//     Drive/Outputs/Out/nCtrl1 @bit 2 <-> STM Control/Control/Reduce torque
//     Drive/Outputs/Out/nCtrl1 @bit 1 <-> STM Control/Control/Reset
//     Drive/Outputs/Out/nDataOut2[0] <-> STM Velocity/Velocity
//   (this object) <-> Device 1 (EtherCAT)/Power (EK1200)/PLC Junction 2 (EK1122)/PLC Coupler 2 (EK1100)/PLC Junction 10 (EK1122)/Granite3 (EK1100)/PLC Junction 12  (EK1122)/TM2K4 (EK1100)/TM2K4-EL5042-E3
//     Enc/Inputs/In/nComState @bit 1 <-> WcState/InputToggle
//     Enc/Inputs/In/nComState <-> WcState/WcState
//     Enc/Inputs/In/nDataIn1 <-> FB Inputs Channel 1/Position
//     Enc/Inputs/In/nDataIn1 <-> FB Inputs Channel 2/Position
//     Enc/Inputs/In/nState1 @bit 12 <-> FB Inputs Channel 1/Status/Diag
//     Enc/Inputs/In/nState1 @bit 12 <-> FB Inputs Channel 2/Status/Diag
//     Enc/Inputs/In/nState1 @bit 1 <-> FB Inputs Channel 1/Status/Error
//     Enc/Inputs/In/nState1 @bit 1 <-> FB Inputs Channel 2/Status/Error
//     Enc/Inputs/In/nState1 @bit 14 <-> FB Inputs Channel 1/Status/Input cycle counter
//     Enc/Inputs/In/nState1 @bit 14 <-> FB Inputs Channel 2/Status/Input cycle counter
//     Enc/Inputs/In/nState1 @bit 2 <-> FB Inputs Channel 1/Status/Ready
//     Enc/Inputs/In/nState1 @bit 2 <-> FB Inputs Channel 2/Status/Ready
//     Enc/Inputs/In/nState1 @bit 13 <-> FB Inputs Channel 1/Status/TxPDO State
//     Enc/Inputs/In/nState1 @bit 13 <-> FB Inputs Channel 2/Status/TxPDO State
//     Enc/Inputs/In/nState1 <-> FB Inputs Channel 1/Status/Warning
//     Enc/Inputs/In/nState1 <-> FB Inputs Channel 2/Status/Warning
//   (this object) <-> Device 1 (EtherCAT)/Power (EK1200)/PLC Junction 2 (EK1122)/PLC Coupler 2 (EK1100)/PLC Junction 10 (EK1122)/Granite3 (EK1100)/PLC Junction 12  (EK1122)/TM2K4 (EK1100)/TM2K4-EL7041-E1
//     Drive/Inputs/In/nState1 @bit 3 <-> STM Status/Status/Error
//     Drive/Inputs/In/nState1 @bit 5 <-> STM Status/Status/Moving negative
//     Drive/Inputs/In/nState1 @bit 4 <-> STM Status/Status/Moving positive
//     Drive/Inputs/In/nState1 @bit 1 <-> STM Status/Status/Ready
//     Drive/Inputs/In/nState1 <-> STM Status/Status/Ready to enable
//     Drive/Inputs/In/nState1 @bit 6 <-> STM Status/Status/Torque reduced
//     Drive/Inputs/In/nState1 @bit 2 <-> STM Status/Status/Warning
//     Drive/Inputs/In/nState2 @bit 3 <-> STM Status/Status/Digital input 1
//     Drive/Inputs/In/nState2 @bit 4 <-> STM Status/Status/Digital input 2
//     Drive/Inputs/In/nState2 @bit 5 <-> STM Status/Status/Sync error
//     Drive/Inputs/In/nState2 @bit 7 <-> STM Status/Status/TxPDO Toggle
//     Drive/Inputs/In/nState4 @bit 1 <-> WcState/InputToggle
//     Drive/Inputs/In/nState4 <-> WcState/WcState
//     Drive/Outputs/Out/nCtrl1 <-> STM Control/Control/Enable
//     Drive/Outputs/Out/nCtrl1 @bit 2 <-> STM Control/Control/Reduce torque
//     Drive/Outputs/Out/nCtrl1 @bit 1 <-> STM Control/Control/Reset
//     Drive/Outputs/Out/nDataOut2[0] <-> STM Velocity/Velocity
//   (this object) <-> Device 1 (EtherCAT)/Power (EK1200)/PLC Junction 2 (EK1122)/PLC Coupler 2 (EK1100)/PLC Junction 10 (EK1122)/Granite3 (EK1100)/PLC Junction 12  (EK1122)/TM2K4 (EK1100)/TM2K4-EL7041-E2
//     Drive/Inputs/In/nState1 @bit 3 <-> STM Status/Status/Error
//     Drive/Inputs/In/nState1 @bit 5 <-> STM Status/Status/Moving negative
//     Drive/Inputs/In/nState1 @bit 4 <-> STM Status/Status/Moving positive
//     Drive/Inputs/In/nState1 @bit 1 <-> STM Status/Status/Ready
//     Drive/Inputs/In/nState1 <-> STM Status/Status/Ready to enable
//     Drive/Inputs/In/nState1 @bit 6 <-> STM Status/Status/Torque reduced
//     Drive/Inputs/In/nState1 @bit 2 <-> STM Status/Status/Warning
//     Drive/Inputs/In/nState2 @bit 3 <-> STM Status/Status/Digital input 1
//     Drive/Inputs/In/nState2 @bit 4 <-> STM Status/Status/Digital input 2
//     Drive/Inputs/In/nState2 @bit 5 <-> STM Status/Status/Sync error
//     Drive/Inputs/In/nState2 @bit 7 <-> STM Status/Status/TxPDO Toggle
//     Drive/Inputs/In/nState4 @bit 1 <-> WcState/InputToggle
//     Drive/Inputs/In/nState4 <-> WcState/WcState
//     Drive/Outputs/Out/nCtrl1 <-> STM Control/Control/Enable
//     Drive/Outputs/Out/nCtrl1 @bit 2 <-> STM Control/Control/Reduce torque
//     Drive/Outputs/Out/nCtrl1 @bit 1 <-> STM Control/Control/Reset
//     Drive/Outputs/Out/nDataOut2[0] <-> STM Velocity/Velocity
//   (this object) <-> Device 1 (EtherCAT)/Power (EK1200)/PLC Junction 2 (EK1122)/PLC Coupler 2 (EK1100)/PLC Junction 10 (EK1122)/Granite3 (EK1100)/PLC Junction 12  (EK1122)/IM6K4 (EK1100)/IM6K4-EL5042-E2
//     Enc/Inputs/In/nComState @bit 1 <-> WcState/InputToggle
//     Enc/Inputs/In/nComState <-> WcState/WcState
//     Enc/Inputs/In/nDataIn1 <-> FB Inputs Channel 1/Position
//     Enc/Inputs/In/nState1 @bit 12 <-> FB Inputs Channel 1/Status/Diag
//     Enc/Inputs/In/nState1 @bit 1 <-> FB Inputs Channel 1/Status/Error
//     Enc/Inputs/In/nState1 @bit 14 <-> FB Inputs Channel 1/Status/Input cycle counter
//     Enc/Inputs/In/nState1 @bit 2 <-> FB Inputs Channel 1/Status/Ready
//     Enc/Inputs/In/nState1 @bit 13 <-> FB Inputs Channel 1/Status/TxPDO State
//     Enc/Inputs/In/nState1 <-> FB Inputs Channel 1/Status/Warning
//   (this object) <-> Device 1 (EtherCAT)/Power (EK1200)/PLC Junction 2 (EK1122)/PLC Coupler 2 (EK1100)/PLC Junction 10 (EK1122)/Granite3 (EK1100)/PLC Junction 12  (EK1122)/IM6K4 (EK1100)/IM6K4-EL7041-E1
//     Drive/Inputs/In/nState1 @bit 3 <-> STM Status/Status/Error
//     Drive/Inputs/In/nState1 @bit 5 <-> STM Status/Status/Moving negative
//     Drive/Inputs/In/nState1 @bit 4 <-> STM Status/Status/Moving positive
//     Drive/Inputs/In/nState1 @bit 1 <-> STM Status/Status/Ready
//     Drive/Inputs/In/nState1 <-> STM Status/Status/Ready to enable
//     Drive/Inputs/In/nState1 @bit 6 <-> STM Status/Status/Torque reduced
//     Drive/Inputs/In/nState1 @bit 2 <-> STM Status/Status/Warning
//     Drive/Inputs/In/nState2 @bit 3 <-> STM Status/Status/Digital input 1
//     Drive/Inputs/In/nState2 @bit 4 <-> STM Status/Status/Digital input 2
//     Drive/Inputs/In/nState2 @bit 5 <-> STM Status/Status/Sync error
//     Drive/Inputs/In/nState2 @bit 7 <-> STM Status/Status/TxPDO Toggle
//     Drive/Inputs/In/nState4 @bit 1 <-> WcState/InputToggle
//     Drive/Inputs/In/nState4 <-> WcState/WcState
//     Drive/Outputs/Out/nCtrl1 <-> STM Control/Control/Enable
//     Drive/Outputs/Out/nCtrl1 @bit 2 <-> STM Control/Control/Reduce torque
//     Drive/Outputs/Out/nCtrl1 @bit 1 <-> STM Control/Control/Reset
//     Drive/Outputs/Out/nDataOut2[0] <-> STM Velocity/Velocity
//   (this object) <-> Device 1 (EtherCAT)/Power (EK1200)/PLC Junction 2 (EK1122)/PLC Coupler 2 (EK1100)/PLC Junction 10 (EK1122)/Granite3 (EK1100)/PLC Junction 11 (EK1122)/PF2K4-WFS (EK1100)/PF2K4-EL5042-E3
//     Enc/Inputs/In/nComState @bit 1 <-> WcState/InputToggle
//     Enc/Inputs/In/nComState <-> WcState/WcState
//     Enc/Inputs/In/nDataIn1 <-> FB Inputs Channel 2/Position
//     Enc/Inputs/In/nDataIn1 <-> FB Inputs Channel 1/Position
//     Enc/Inputs/In/nState1 @bit 12 <-> FB Inputs Channel 2/Status/Diag
//     Enc/Inputs/In/nState1 @bit 12 <-> FB Inputs Channel 1/Status/Diag
//     Enc/Inputs/In/nState1 @bit 1 <-> FB Inputs Channel 2/Status/Error
//     Enc/Inputs/In/nState1 @bit 1 <-> FB Inputs Channel 1/Status/Error
//     Enc/Inputs/In/nState1 @bit 14 <-> FB Inputs Channel 2/Status/Input cycle counter
//     Enc/Inputs/In/nState1 @bit 14 <-> FB Inputs Channel 1/Status/Input cycle counter
//     Enc/Inputs/In/nState1 @bit 2 <-> FB Inputs Channel 2/Status/Ready
//     Enc/Inputs/In/nState1 @bit 2 <-> FB Inputs Channel 1/Status/Ready
//     Enc/Inputs/In/nState1 @bit 13 <-> FB Inputs Channel 2/Status/TxPDO State
//     Enc/Inputs/In/nState1 @bit 13 <-> FB Inputs Channel 1/Status/TxPDO State
//     Enc/Inputs/In/nState1 <-> FB Inputs Channel 2/Status/Warning
//     Enc/Inputs/In/nState1 <-> FB Inputs Channel 1/Status/Warning
//   (this object) <-> Device 1 (EtherCAT)/Power (EK1200)/PLC Junction 2 (EK1122)/PLC Coupler 2 (EK1100)/PLC Junction 10 (EK1122)/Granite3 (EK1100)/PLC Junction 11 (EK1122)/PF2K4-WFS (EK1100)/PF2K4-EL7041-E1
//     Drive/Inputs/In/nState1 @bit 3 <-> STM Status/Status/Error
//     Drive/Inputs/In/nState1 @bit 5 <-> STM Status/Status/Moving negative
//     Drive/Inputs/In/nState1 @bit 4 <-> STM Status/Status/Moving positive
//     Drive/Inputs/In/nState1 @bit 1 <-> STM Status/Status/Ready
//     Drive/Inputs/In/nState1 <-> STM Status/Status/Ready to enable
//     Drive/Inputs/In/nState1 @bit 6 <-> STM Status/Status/Torque reduced
//     Drive/Inputs/In/nState1 @bit 2 <-> STM Status/Status/Warning
//     Drive/Inputs/In/nState2 @bit 3 <-> STM Status/Status/Digital input 1
//     Drive/Inputs/In/nState2 @bit 4 <-> STM Status/Status/Digital input 2
//     Drive/Inputs/In/nState2 @bit 5 <-> STM Status/Status/Sync error
//     Drive/Inputs/In/nState2 @bit 7 <-> STM Status/Status/TxPDO Toggle
//     Drive/Inputs/In/nState4 @bit 1 <-> WcState/InputToggle
//     Drive/Inputs/In/nState4 <-> WcState/WcState
//     Drive/Outputs/Out/nCtrl1 <-> STM Control/Control/Enable
//     Drive/Outputs/Out/nCtrl1 @bit 2 <-> STM Control/Control/Reduce torque
//     Drive/Outputs/Out/nCtrl1 @bit 1 <-> STM Control/Control/Reset
//     Drive/Outputs/Out/nDataOut2[0] <-> STM Velocity/Velocity
//   (this object) <-> Device 1 (EtherCAT)/Power (EK1200)/PLC Junction 2 (EK1122)/PLC Coupler 2 (EK1100)/PLC Junction 10 (EK1122)/Granite3 (EK1100)/PLC Junction 11 (EK1122)/PF2K4-WFS (EK1100)/PF2K4-EL7041-E2
//     Drive/Inputs/In/nState1 @bit 3 <-> STM Status/Status/Error
//     Drive/Inputs/In/nState1 @bit 5 <-> STM Status/Status/Moving negative
//     Drive/Inputs/In/nState1 @bit 4 <-> STM Status/Status/Moving positive
//     Drive/Inputs/In/nState1 @bit 1 <-> STM Status/Status/Ready
//     Drive/Inputs/In/nState1 <-> STM Status/Status/Ready to enable
//     Drive/Inputs/In/nState1 @bit 6 <-> STM Status/Status/Torque reduced
//     Drive/Inputs/In/nState1 @bit 2 <-> STM Status/Status/Warning
//     Drive/Inputs/In/nState2 @bit 3 <-> STM Status/Status/Digital input 1
//     Drive/Inputs/In/nState2 @bit 4 <-> STM Status/Status/Digital input 2
//     Drive/Inputs/In/nState2 @bit 5 <-> STM Status/Status/Sync error
//     Drive/Inputs/In/nState2 @bit 7 <-> STM Status/Status/TxPDO Toggle
//     Drive/Inputs/In/nState4 @bit 1 <-> WcState/InputToggle
//     Drive/Inputs/In/nState4 <-> WcState/WcState
//     Drive/Outputs/Out/nCtrl1 <-> STM Control/Control/Enable
//     Drive/Outputs/Out/nCtrl1 @bit 2 <-> STM Control/Control/Reduce torque
//     Drive/Outputs/Out/nCtrl1 @bit 1 <-> STM Control/Control/Reset
//     Drive/Outputs/Out/nDataOut2[0] <-> STM Velocity/Velocity
//   (this object) <-> Device 1 (EtherCAT)/Power (EK1200)/PLC Junction 2 (EK1122)/PLC Coupler 2 (EK1100)/PLC Junction 9 (EK1122)/SP1K4 Bottom Rail (EK1100)/EL7031-LensX
//     Drive/Inputs/In/nState1 @bit 3 <-> STM Status/Status/Error
//     Drive/Inputs/In/nState1 @bit 5 <-> STM Status/Status/Moving negative
//     Drive/Inputs/In/nState1 @bit 4 <-> STM Status/Status/Moving positive
//     Drive/Inputs/In/nState1 @bit 1 <-> STM Status/Status/Ready
//     Drive/Inputs/In/nState1 <-> STM Status/Status/Ready to enable
//     Drive/Inputs/In/nState1 @bit 6 <-> STM Status/Status/Torque reduced
//     Drive/Inputs/In/nState1 @bit 2 <-> STM Status/Status/Warning
//     Drive/Inputs/In/nState2 @bit 3 <-> STM Status/Status/Digital input 1
//     Drive/Inputs/In/nState2 @bit 4 <-> STM Status/Status/Digital input 2
//     Drive/Inputs/In/nState2 @bit 5 <-> STM Status/Status/Sync error
//     Drive/Inputs/In/nState2 @bit 7 <-> STM Status/Status/TxPDO Toggle
//     Drive/Inputs/In/nState4 @bit 1 <-> WcState/InputToggle
//     Drive/Inputs/In/nState4 <-> WcState/WcState
//     Drive/Outputs/Out/nCtrl1 <-> STM Control/Control/Enable
//     Drive/Outputs/Out/nCtrl1 @bit 2 <-> STM Control/Control/Reduce torque
//     Drive/Outputs/Out/nCtrl1 @bit 1 <-> STM Control/Control/Reset
//     Drive/Outputs/Out/nDataOut2[0] <-> STM Velocity/Velocity
//     Enc/Inputs/In/nDataIn1[0] <-> ENC Status compact/Counter value
//     Enc/Inputs/In/nDataIn2[0] <-> ENC Status compact/Latch value
//     Enc/Inputs/In/nState1 @bit 4 <-> ENC Status compact/Status/Counter overflow
//     Enc/Inputs/In/nState1 @bit 3 <-> ENC Status compact/Status/Counter underflow
//     Enc/Inputs/In/nState1 @bit 1 <-> ENC Status compact/Status/Latch extern valid
//     Enc/Inputs/In/nState1 @bit 2 <-> ENC Status compact/Status/Set counter done
//     Enc/Inputs/In/nState2 @bit 4 <-> ENC Status compact/Status/Status of extern latch
//     Enc/Inputs/In/nState2 @bit 5 <-> ENC Status compact/Status/Sync error
//     Enc/Inputs/In/nState2 @bit 7 <-> ENC Status compact/Status/TxPDO Toggle
//     Enc/Inputs/In/nState4 @bit 1 <-> WcState/InputToggle
//     Enc/Inputs/In/nState4 <-> WcState/WcState
//     Enc/Outputs/Out/nCtrl1 @bit 3 <-> ENC Control compact/Control/Enable latch extern on negative edge
//     Enc/Outputs/Out/nCtrl1 @bit 1 <-> ENC Control compact/Control/Enable latch extern on positive edge
//     Enc/Outputs/Out/nCtrl1 @bit 2 <-> ENC Control compact/Control/Set counter
//     Enc/Outputs/Out/nDataOut1[0] <-> ENC Control compact/Set counter value
//   (this object) <-> Device 1 (EtherCAT)/Power (EK1200)/PLC Junction 2 (EK1122)/PLC Coupler 2 (EK1100)/PLC Junction 9 (EK1122)/SP1K4 Bottom Rail (EK1100)/FoilX-EL7041
//     Drive/Inputs/In/nState1 @bit 3 <-> STM Status/Status/Error
//     Drive/Inputs/In/nState1 @bit 5 <-> STM Status/Status/Moving negative
//     Drive/Inputs/In/nState1 @bit 4 <-> STM Status/Status/Moving positive
//     Drive/Inputs/In/nState1 @bit 1 <-> STM Status/Status/Ready
//     Drive/Inputs/In/nState1 <-> STM Status/Status/Ready to enable
//     Drive/Inputs/In/nState1 @bit 6 <-> STM Status/Status/Torque reduced
//     Drive/Inputs/In/nState1 @bit 2 <-> STM Status/Status/Warning
//     Drive/Inputs/In/nState2 @bit 3 <-> STM Status/Status/Digital input 1
//     Drive/Inputs/In/nState2 @bit 4 <-> STM Status/Status/Digital input 2
//     Drive/Inputs/In/nState2 @bit 5 <-> STM Status/Status/Sync error
//     Drive/Inputs/In/nState2 @bit 7 <-> STM Status/Status/TxPDO Toggle
//     Drive/Inputs/In/nState4 @bit 1 <-> WcState/InputToggle
//     Drive/Inputs/In/nState4 <-> WcState/WcState
//     Drive/Outputs/Out/nCtrl1 <-> STM Control/Control/Enable
//     Drive/Outputs/Out/nCtrl1 @bit 2 <-> STM Control/Control/Reduce torque
//     Drive/Outputs/Out/nCtrl1 @bit 1 <-> STM Control/Control/Reset
//     Drive/Outputs/Out/nDataOut2[0] <-> STM Velocity/Velocity
//   (this object) <-> Device 1 (EtherCAT)/Power (EK1200)/PLC Junction 2 (EK1122)/PLC Coupler 2 (EK1100)/PLC Junction 9 (EK1122)/SP1K4 Top Rail (EK1100)/SP1K4-EL5042-E2
//     Enc/Inputs/In/nComState @bit 1 <-> WcState/InputToggle
//     Enc/Inputs/In/nComState <-> WcState/WcState
//     Enc/Inputs/In/nDataIn1 <-> FB Inputs Channel 2/Position
//     Enc/Inputs/In/nDataIn1 <-> FB Inputs Channel 1/Position
//     Enc/Inputs/In/nState1 @bit 12 <-> FB Inputs Channel 2/Status/Diag
//     Enc/Inputs/In/nState1 @bit 12 <-> FB Inputs Channel 1/Status/Diag
//     Enc/Inputs/In/nState1 @bit 1 <-> FB Inputs Channel 2/Status/Error
//     Enc/Inputs/In/nState1 @bit 1 <-> FB Inputs Channel 1/Status/Error
//     Enc/Inputs/In/nState1 @bit 14 <-> FB Inputs Channel 2/Status/Input cycle counter
//     Enc/Inputs/In/nState1 @bit 14 <-> FB Inputs Channel 1/Status/Input cycle counter
//     Enc/Inputs/In/nState1 @bit 2 <-> FB Inputs Channel 2/Status/Ready
//     Enc/Inputs/In/nState1 @bit 2 <-> FB Inputs Channel 1/Status/Ready
//     Enc/Inputs/In/nState1 @bit 13 <-> FB Inputs Channel 2/Status/TxPDO State
//     Enc/Inputs/In/nState1 @bit 13 <-> FB Inputs Channel 1/Status/TxPDO State
//     Enc/Inputs/In/nState1 <-> FB Inputs Channel 2/Status/Warning
//     Enc/Inputs/In/nState1 <-> FB Inputs Channel 1/Status/Warning
//   (this object) <-> Device 1 (EtherCAT)/Power (EK1200)/PLC Junction 2 (EK1122)/PLC Coupler 2 (EK1100)/PLC Junction 9 (EK1122)/SP1K4 Bottom Rail (EK1100)/ZonePlateX-EL7041
//     Drive/Inputs/In/nState1 @bit 3 <-> STM Status/Status/Error
//     Drive/Inputs/In/nState1 @bit 5 <-> STM Status/Status/Moving negative
//     Drive/Inputs/In/nState1 @bit 4 <-> STM Status/Status/Moving positive
//     Drive/Inputs/In/nState1 @bit 1 <-> STM Status/Status/Ready
//     Drive/Inputs/In/nState1 <-> STM Status/Status/Ready to enable
//     Drive/Inputs/In/nState1 @bit 6 <-> STM Status/Status/Torque reduced
//     Drive/Inputs/In/nState1 @bit 2 <-> STM Status/Status/Warning
//     Drive/Inputs/In/nState2 @bit 3 <-> STM Status/Status/Digital input 1
//     Drive/Inputs/In/nState2 @bit 4 <-> STM Status/Status/Digital input 2
//     Drive/Inputs/In/nState2 @bit 5 <-> STM Status/Status/Sync error
//     Drive/Inputs/In/nState2 @bit 7 <-> STM Status/Status/TxPDO Toggle
//     Drive/Inputs/In/nState4 @bit 1 <-> WcState/InputToggle
//     Drive/Inputs/In/nState4 <-> WcState/WcState
//     Drive/Outputs/Out/nCtrl1 <-> STM Control/Control/Enable
//     Drive/Outputs/Out/nCtrl1 @bit 2 <-> STM Control/Control/Reduce torque
//     Drive/Outputs/Out/nCtrl1 @bit 1 <-> STM Control/Control/Reset
//     Drive/Outputs/Out/nDataOut2[0] <-> STM Velocity/Velocity
//   (this object) <-> Device 1 (EtherCAT)/Power (EK1200)/PLC Junction 2 (EK1122)/PLC Coupler 2 (EK1100)/PLC Junction 9 (EK1122)/SP1K4 Top Rail (EK1100)/SP1K4-EL5042-E1
//     Enc/Inputs/In/nComState @bit 1 <-> WcState/InputToggle
//     Enc/Inputs/In/nComState <-> WcState/WcState
//     Enc/Inputs/In/nDataIn1 <-> FB Inputs Channel 1/Position
//     Enc/Inputs/In/nDataIn1 <-> FB Inputs Channel 2/Position
//     Enc/Inputs/In/nState1 @bit 12 <-> FB Inputs Channel 1/Status/Diag
//     Enc/Inputs/In/nState1 @bit 12 <-> FB Inputs Channel 2/Status/Diag
//     Enc/Inputs/In/nState1 @bit 1 <-> FB Inputs Channel 1/Status/Error
//     Enc/Inputs/In/nState1 @bit 1 <-> FB Inputs Channel 2/Status/Error
//     Enc/Inputs/In/nState1 @bit 14 <-> FB Inputs Channel 1/Status/Input cycle counter
//     Enc/Inputs/In/nState1 @bit 14 <-> FB Inputs Channel 2/Status/Input cycle counter
//     Enc/Inputs/In/nState1 @bit 2 <-> FB Inputs Channel 1/Status/Ready
//     Enc/Inputs/In/nState1 @bit 2 <-> FB Inputs Channel 2/Status/Ready
//     Enc/Inputs/In/nState1 @bit 13 <-> FB Inputs Channel 1/Status/TxPDO State
//     Enc/Inputs/In/nState1 @bit 13 <-> FB Inputs Channel 2/Status/TxPDO State
//     Enc/Inputs/In/nState1 <-> FB Inputs Channel 1/Status/Warning
//     Enc/Inputs/In/nState1 <-> FB Inputs Channel 2/Status/Warning
//   (this object) <-> Device 1 (EtherCAT)/Power (EK1200)/PLC Junction 2 (EK1122)/PLC Coupler 2 (EK1100)/PLC Junction 9 (EK1122)/SP1K4 Bottom Rail (EK1100)/ZonePlateY-EL7041
//     Drive/Inputs/In/nState1 @bit 3 <-> STM Status/Status/Error
//     Drive/Inputs/In/nState1 @bit 5 <-> STM Status/Status/Moving negative
//     Drive/Inputs/In/nState1 @bit 4 <-> STM Status/Status/Moving positive
//     Drive/Inputs/In/nState1 @bit 1 <-> STM Status/Status/Ready
//     Drive/Inputs/In/nState1 <-> STM Status/Status/Ready to enable
//     Drive/Inputs/In/nState1 @bit 6 <-> STM Status/Status/Torque reduced
//     Drive/Inputs/In/nState1 @bit 2 <-> STM Status/Status/Warning
//     Drive/Inputs/In/nState2 @bit 3 <-> STM Status/Status/Digital input 1
//     Drive/Inputs/In/nState2 @bit 4 <-> STM Status/Status/Digital input 2
//     Drive/Inputs/In/nState2 @bit 5 <-> STM Status/Status/Sync error
//     Drive/Inputs/In/nState2 @bit 7 <-> STM Status/Status/TxPDO Toggle
//     Drive/Inputs/In/nState4 @bit 1 <-> WcState/InputToggle
//     Drive/Inputs/In/nState4 <-> WcState/WcState
//     Drive/Outputs/Out/nCtrl1 <-> STM Control/Control/Enable
//     Drive/Outputs/Out/nCtrl1 @bit 2 <-> STM Control/Control/Reduce torque
//     Drive/Outputs/Out/nCtrl1 @bit 1 <-> STM Control/Control/Reset
//     Drive/Outputs/Out/nDataOut2[0] <-> STM Velocity/Velocity
//   (this object) <-> Device 1 (EtherCAT)/Power (EK1200)/PLC Junction 2 (EK1122)/PLC Coupler 2 (EK1100)/PLC Junction 9 (EK1122)/SP1K4 Bottom Rail (EK1100)/ZonePlateZ-EL7041
//     Drive/Inputs/In/nState1 @bit 3 <-> STM Status/Status/Error
//     Drive/Inputs/In/nState1 @bit 5 <-> STM Status/Status/Moving negative
//     Drive/Inputs/In/nState1 @bit 4 <-> STM Status/Status/Moving positive
//     Drive/Inputs/In/nState1 @bit 1 <-> STM Status/Status/Ready
//     Drive/Inputs/In/nState1 <-> STM Status/Status/Ready to enable
//     Drive/Inputs/In/nState1 @bit 6 <-> STM Status/Status/Torque reduced
//     Drive/Inputs/In/nState1 @bit 2 <-> STM Status/Status/Warning
//     Drive/Inputs/In/nState2 @bit 3 <-> STM Status/Status/Digital input 1
//     Drive/Inputs/In/nState2 @bit 4 <-> STM Status/Status/Digital input 2
//     Drive/Inputs/In/nState2 @bit 5 <-> STM Status/Status/Sync error
//     Drive/Inputs/In/nState2 @bit 7 <-> STM Status/Status/TxPDO Toggle
//     Drive/Inputs/In/nState4 @bit 1 <-> WcState/InputToggle
//     Drive/Inputs/In/nState4 <-> WcState/WcState
//     Drive/Outputs/Out/nCtrl1 <-> STM Control/Control/Enable
//     Drive/Outputs/Out/nCtrl1 @bit 2 <-> STM Control/Control/Reduce torque
//     Drive/Outputs/Out/nCtrl1 @bit 1 <-> STM Control/Control/Reset
//     Drive/Outputs/Out/nDataOut2[0] <-> STM Velocity/Velocity
//   (this object) <-> Device 1 (EtherCAT)/Power (EK1200)/PLC Junction 2 (EK1122)/PLC Coupler 2 (EK1100)/PLC Junction 9 (EK1122)/SP1K4 Bottom Rail (EK1100)/YagX-EL7041
//     Drive/Inputs/In/nState1 @bit 3 <-> STM Status/Status/Error
//     Drive/Inputs/In/nState1 @bit 5 <-> STM Status/Status/Moving negative
//     Drive/Inputs/In/nState1 @bit 4 <-> STM Status/Status/Moving positive
//     Drive/Inputs/In/nState1 @bit 1 <-> STM Status/Status/Ready
//     Drive/Inputs/In/nState1 <-> STM Status/Status/Ready to enable
//     Drive/Inputs/In/nState1 @bit 6 <-> STM Status/Status/Torque reduced
//     Drive/Inputs/In/nState1 @bit 2 <-> STM Status/Status/Warning
//     Drive/Inputs/In/nState2 @bit 3 <-> STM Status/Status/Digital input 1
//     Drive/Inputs/In/nState2 @bit 4 <-> STM Status/Status/Digital input 2
//     Drive/Inputs/In/nState2 @bit 5 <-> STM Status/Status/Sync error
//     Drive/Inputs/In/nState2 @bit 7 <-> STM Status/Status/TxPDO Toggle
//     Drive/Inputs/In/nState4 @bit 1 <-> WcState/InputToggle
//     Drive/Inputs/In/nState4 <-> WcState/WcState
//     Drive/Outputs/Out/nCtrl1 <-> STM Control/Control/Enable
//     Drive/Outputs/Out/nCtrl1 @bit 2 <-> STM Control/Control/Reduce torque
//     Drive/Outputs/Out/nCtrl1 @bit 1 <-> STM Control/Control/Reset
//     Drive/Outputs/Out/nDataOut2[0] <-> STM Velocity/Velocity
//   (this object) <-> Device 1 (EtherCAT)/Power (EK1200)/PLC Junction 2 (EK1122)/PLC Coupler 2 (EK1100)/PLC Junction 9 (EK1122)/SP1K4 Top Rail (EK1100)/SP1K4-EL5042-E8
//     Enc/Inputs/In/nComState @bit 1 <-> WcState/InputToggle
//     Enc/Inputs/In/nComState <-> WcState/WcState
//     Enc/Inputs/In/nDataIn1 <-> FB Inputs Channel 1/Position
//     Enc/Inputs/In/nDataIn1 <-> FB Inputs Channel 2/Position
//     Enc/Inputs/In/nState1 @bit 12 <-> FB Inputs Channel 1/Status/Diag
//     Enc/Inputs/In/nState1 @bit 12 <-> FB Inputs Channel 2/Status/Diag
//     Enc/Inputs/In/nState1 @bit 1 <-> FB Inputs Channel 1/Status/Error
//     Enc/Inputs/In/nState1 @bit 1 <-> FB Inputs Channel 2/Status/Error
//     Enc/Inputs/In/nState1 @bit 14 <-> FB Inputs Channel 1/Status/Input cycle counter
//     Enc/Inputs/In/nState1 @bit 14 <-> FB Inputs Channel 2/Status/Input cycle counter
//     Enc/Inputs/In/nState1 @bit 2 <-> FB Inputs Channel 1/Status/Ready
//     Enc/Inputs/In/nState1 @bit 2 <-> FB Inputs Channel 2/Status/Ready
//     Enc/Inputs/In/nState1 @bit 13 <-> FB Inputs Channel 1/Status/TxPDO State
//     Enc/Inputs/In/nState1 @bit 13 <-> FB Inputs Channel 2/Status/TxPDO State
//     Enc/Inputs/In/nState1 <-> FB Inputs Channel 1/Status/Warning
//     Enc/Inputs/In/nState1 <-> FB Inputs Channel 2/Status/Warning
//   (this object) <-> Device 1 (EtherCAT)/Power (EK1200)/PLC Junction 2 (EK1122)/PLC Coupler 2 (EK1100)/PLC Junction 9 (EK1122)/SP1K4 Bottom Rail (EK1100)/YagY-EL7041
//     Drive/Inputs/In/nState1 @bit 3 <-> STM Status/Status/Error
//     Drive/Inputs/In/nState1 @bit 5 <-> STM Status/Status/Moving negative
//     Drive/Inputs/In/nState1 @bit 4 <-> STM Status/Status/Moving positive
//     Drive/Inputs/In/nState1 @bit 1 <-> STM Status/Status/Ready
//     Drive/Inputs/In/nState1 <-> STM Status/Status/Ready to enable
//     Drive/Inputs/In/nState1 @bit 6 <-> STM Status/Status/Torque reduced
//     Drive/Inputs/In/nState1 @bit 2 <-> STM Status/Status/Warning
//     Drive/Inputs/In/nState2 @bit 3 <-> STM Status/Status/Digital input 1
//     Drive/Inputs/In/nState2 @bit 4 <-> STM Status/Status/Digital input 2
//     Drive/Inputs/In/nState2 @bit 5 <-> STM Status/Status/Sync error
//     Drive/Inputs/In/nState2 @bit 7 <-> STM Status/Status/TxPDO Toggle
//     Drive/Inputs/In/nState4 @bit 1 <-> WcState/InputToggle
//     Drive/Inputs/In/nState4 <-> WcState/WcState
//     Drive/Outputs/Out/nCtrl1 <-> STM Control/Control/Enable
//     Drive/Outputs/Out/nCtrl1 @bit 2 <-> STM Control/Control/Reduce torque
//     Drive/Outputs/Out/nCtrl1 @bit 1 <-> STM Control/Control/Reset
//     Drive/Outputs/Out/nDataOut2[0] <-> STM Velocity/Velocity
//     Enc/Inputs/In/nDataIn1[0] <-> ENC Status compact/Counter value
//     Enc/Inputs/In/nDataIn2[0] <-> ENC Status compact/Latch value
//     Enc/Inputs/In/nState1 @bit 4 <-> ENC Status compact/Status/Counter overflow
//     Enc/Inputs/In/nState1 @bit 3 <-> ENC Status compact/Status/Counter underflow
//     Enc/Inputs/In/nState1 @bit 7 <-> ENC Status compact/Status/Extrapolation stall
//     Enc/Inputs/In/nState1 <-> ENC Status compact/Status/Latch C valid
//     Enc/Inputs/In/nState1 @bit 1 <-> ENC Status compact/Status/Latch extern valid
//     Enc/Inputs/In/nState1 @bit 2 <-> ENC Status compact/Status/Set counter done
//     Enc/Inputs/In/nState2 @bit 4 <-> ENC Status compact/Status/Status of extern latch
//     Enc/Inputs/In/nState2 <-> ENC Status compact/Status/Status of input A
//     Enc/Inputs/In/nState2 @bit 1 <-> ENC Status compact/Status/Status of input B
//     Enc/Inputs/In/nState2 @bit 2 <-> ENC Status compact/Status/Status of input C
//     Enc/Inputs/In/nState2 @bit 5 <-> ENC Status compact/Status/Sync error
//     Enc/Inputs/In/nState2 @bit 7 <-> ENC Status compact/Status/TxPDO Toggle
//     Enc/Inputs/In/nState4 @bit 1 <-> WcState/InputToggle
//     Enc/Inputs/In/nState4 <-> WcState/WcState
//     Enc/Outputs/Out/nCtrl1 <-> ENC Control compact/Control/Enable latch C
//     Enc/Outputs/Out/nCtrl1 @bit 3 <-> ENC Control compact/Control/Enable latch extern on negative edge
//     Enc/Outputs/Out/nCtrl1 @bit 1 <-> ENC Control compact/Control/Enable latch extern on positive edge
//     Enc/Outputs/Out/nCtrl1 @bit 2 <-> ENC Control compact/Control/Set counter
//     Enc/Outputs/Out/nDataOut1[0] <-> ENC Control compact/Set counter value
//   (this object) <-> Device 1 (EtherCAT)/Power (EK1200)/PLC Junction 2 (EK1122)/PLC Coupler 2 (EK1100)/PLC Junction 9 (EK1122)/SP1K4 Bottom Rail (EK1100)/YagZ-EL7041
//     Drive/Inputs/In/nState1 @bit 3 <-> STM Status/Status/Error
//     Drive/Inputs/In/nState1 @bit 5 <-> STM Status/Status/Moving negative
//     Drive/Inputs/In/nState1 @bit 4 <-> STM Status/Status/Moving positive
//     Drive/Inputs/In/nState1 @bit 1 <-> STM Status/Status/Ready
//     Drive/Inputs/In/nState1 <-> STM Status/Status/Ready to enable
//     Drive/Inputs/In/nState1 @bit 6 <-> STM Status/Status/Torque reduced
//     Drive/Inputs/In/nState1 @bit 2 <-> STM Status/Status/Warning
//     Drive/Inputs/In/nState2 @bit 3 <-> STM Status/Status/Digital input 1
//     Drive/Inputs/In/nState2 @bit 4 <-> STM Status/Status/Digital input 2
//     Drive/Inputs/In/nState2 @bit 5 <-> STM Status/Status/Sync error
//     Drive/Inputs/In/nState2 @bit 7 <-> STM Status/Status/TxPDO Toggle
//     Drive/Inputs/In/nState4 @bit 1 <-> WcState/InputToggle
//     Drive/Inputs/In/nState4 <-> WcState/WcState
//     Drive/Outputs/Out/nCtrl1 <-> STM Control/Control/Enable
//     Drive/Outputs/Out/nCtrl1 @bit 2 <-> STM Control/Control/Reduce torque
//     Drive/Outputs/Out/nCtrl1 @bit 1 <-> STM Control/Control/Reset
//     Drive/Outputs/Out/nDataOut2[0] <-> STM Velocity/Velocity
//   (this object) <-> Device 1 (EtherCAT)/Power (EK1200)/PLC Junction 2 (EK1122)/PLC Coupler 2 (EK1100)/PLC Junction 9 (EK1122)/SP1K4 Bottom Rail (EK1100)/YagTheta-EL7041
//     Drive/Inputs/In/nState1 @bit 3 <-> STM Status/Status/Error
//     Drive/Inputs/In/nState1 @bit 5 <-> STM Status/Status/Moving negative
//     Drive/Inputs/In/nState1 @bit 4 <-> STM Status/Status/Moving positive
//     Drive/Inputs/In/nState1 @bit 1 <-> STM Status/Status/Ready
//     Drive/Inputs/In/nState1 <-> STM Status/Status/Ready to enable
//     Drive/Inputs/In/nState1 @bit 6 <-> STM Status/Status/Torque reduced
//     Drive/Inputs/In/nState1 @bit 2 <-> STM Status/Status/Warning
//     Drive/Inputs/In/nState2 @bit 3 <-> STM Status/Status/Digital input 1
//     Drive/Inputs/In/nState2 @bit 4 <-> STM Status/Status/Digital input 2
//     Drive/Inputs/In/nState2 @bit 5 <-> STM Status/Status/Sync error
//     Drive/Inputs/In/nState2 @bit 7 <-> STM Status/Status/TxPDO Toggle
//     Drive/Inputs/In/nState4 @bit 1 <-> WcState/InputToggle
//     Drive/Inputs/In/nState4 <-> WcState/WcState
//     Drive/Outputs/Out/nCtrl1 <-> STM Control/Control/Enable
//     Drive/Outputs/Out/nCtrl1 @bit 2 <-> STM Control/Control/Reduce torque
//     Drive/Outputs/Out/nCtrl1 @bit 1 <-> STM Control/Control/Reset
//     Drive/Outputs/Out/nDataOut2[0] <-> STM Velocity/Velocity
//     Enc/Inputs/In/nDataIn1[0] <-> ENC Status compact/Counter value
//     Enc/Inputs/In/nDataIn2[0] <-> ENC Status compact/Latch value
//     Enc/Inputs/In/nState1 @bit 4 <-> ENC Status compact/Status/Counter overflow
//     Enc/Inputs/In/nState1 @bit 3 <-> ENC Status compact/Status/Counter underflow
//     Enc/Inputs/In/nState1 @bit 7 <-> ENC Status compact/Status/Extrapolation stall
//     Enc/Inputs/In/nState1 <-> ENC Status compact/Status/Latch C valid
//     Enc/Inputs/In/nState1 @bit 1 <-> ENC Status compact/Status/Latch extern valid
//     Enc/Inputs/In/nState1 @bit 2 <-> ENC Status compact/Status/Set counter done
//     Enc/Inputs/In/nState2 @bit 4 <-> ENC Status compact/Status/Status of extern latch
//     Enc/Inputs/In/nState2 <-> ENC Status compact/Status/Status of input A
//     Enc/Inputs/In/nState2 @bit 1 <-> ENC Status compact/Status/Status of input B
//     Enc/Inputs/In/nState2 @bit 2 <-> ENC Status compact/Status/Status of input C
//     Enc/Inputs/In/nState2 @bit 5 <-> ENC Status compact/Status/Sync error
//     Enc/Inputs/In/nState2 @bit 7 <-> ENC Status compact/Status/TxPDO Toggle
//     Enc/Inputs/In/nState4 @bit 1 <-> WcState/InputToggle
//     Enc/Inputs/In/nState4 <-> WcState/WcState
//     Enc/Outputs/Out/nCtrl1 <-> ENC Control compact/Control/Enable latch C
//     Enc/Outputs/Out/nCtrl1 @bit 3 <-> ENC Control compact/Control/Enable latch extern on negative edge
//     Enc/Outputs/Out/nCtrl1 @bit 1 <-> ENC Control compact/Control/Enable latch extern on positive edge
//     Enc/Outputs/Out/nCtrl1 @bit 2 <-> ENC Control compact/Control/Set counter
//     Enc/Outputs/Out/nDataOut1[0] <-> ENC Control compact/Set counter value
//   (this object) <-> Device 1 (EtherCAT)/Power (EK1200)/PLC Junction 2 (EK1122)/PLC Coupler 2 (EK1100)/PLC Junction 9 (EK1122)/SP1K4 Top Rail (EK1100)/Term 9 (EL7041)
//     Drive/Inputs/In/nState1 @bit 3 <-> STM Status/Status/Error
//     Drive/Inputs/In/nState1 @bit 5 <-> STM Status/Status/Moving negative
//     Drive/Inputs/In/nState1 @bit 4 <-> STM Status/Status/Moving positive
//     Drive/Inputs/In/nState1 @bit 1 <-> STM Status/Status/Ready
//     Drive/Inputs/In/nState1 <-> STM Status/Status/Ready to enable
//     Drive/Inputs/In/nState1 @bit 6 <-> STM Status/Status/Torque reduced
//     Drive/Inputs/In/nState1 @bit 2 <-> STM Status/Status/Warning
//     Drive/Inputs/In/nState2 @bit 3 <-> STM Status/Status/Digital input 1
//     Drive/Inputs/In/nState2 @bit 4 <-> STM Status/Status/Digital input 2
//     Drive/Inputs/In/nState2 @bit 5 <-> STM Status/Status/Sync error
//     Drive/Inputs/In/nState2 @bit 7 <-> STM Status/Status/TxPDO Toggle
//     Drive/Inputs/In/nState4 @bit 1 <-> WcState/InputToggle
//     Drive/Inputs/In/nState4 <-> WcState/WcState
//     Drive/Outputs/Out/nCtrl1 <-> STM Control/Control/Enable
//     Drive/Outputs/Out/nCtrl1 @bit 2 <-> STM Control/Control/Reduce torque
//     Drive/Outputs/Out/nCtrl1 @bit 1 <-> STM Control/Control/Reset
//     Drive/Outputs/Out/nDataOut2[0] <-> STM Velocity/Velocity
//     Enc/Inputs/In/nDataIn1[0] <-> ENC Status compact/Counter value
//     Enc/Inputs/In/nDataIn2[0] <-> ENC Status compact/Latch value
//     Enc/Inputs/In/nState1 @bit 4 <-> ENC Status compact/Status/Counter overflow
//     Enc/Inputs/In/nState1 @bit 3 <-> ENC Status compact/Status/Counter underflow
//     Enc/Inputs/In/nState1 @bit 7 <-> ENC Status compact/Status/Extrapolation stall
//     Enc/Inputs/In/nState1 <-> ENC Status compact/Status/Latch C valid
//     Enc/Inputs/In/nState1 @bit 1 <-> ENC Status compact/Status/Latch extern valid
//     Enc/Inputs/In/nState1 @bit 2 <-> ENC Status compact/Status/Set counter done
//     Enc/Inputs/In/nState2 @bit 4 <-> ENC Status compact/Status/Status of extern latch
//     Enc/Inputs/In/nState2 <-> ENC Status compact/Status/Status of input A
//     Enc/Inputs/In/nState2 @bit 1 <-> ENC Status compact/Status/Status of input B
//     Enc/Inputs/In/nState2 @bit 2 <-> ENC Status compact/Status/Status of input C
//     Enc/Inputs/In/nState2 @bit 5 <-> ENC Status compact/Status/Sync error
//     Enc/Inputs/In/nState2 @bit 7 <-> ENC Status compact/Status/TxPDO Toggle
//     Enc/Inputs/In/nState4 @bit 1 <-> WcState/InputToggle
//     Enc/Inputs/In/nState4 <-> WcState/WcState
//     Enc/Outputs/Out/nCtrl1 <-> ENC Control compact/Control/Enable latch C
//     Enc/Outputs/Out/nCtrl1 @bit 3 <-> ENC Control compact/Control/Enable latch extern on negative edge
//     Enc/Outputs/Out/nCtrl1 @bit 1 <-> ENC Control compact/Control/Enable latch extern on positive edge
//     Enc/Outputs/Out/nCtrl1 @bit 2 <-> ENC Control compact/Control/Set counter
//     Enc/Outputs/Out/nDataOut1[0] <-> ENC Control compact/Set counter value
//   (this object) <-> Device 1 (EtherCAT)/Power (EK1200)/PLC Junction 2 (EK1122)/PLC Coupler 2 (EK1100)/PLC Junction 9 (EK1122)/SP1K4 Top Rail (EK1100)/Term 10 (EL7041)
//     Drive/Inputs/In/nState1 @bit 3 <-> STM Status/Status/Error
//     Drive/Inputs/In/nState1 @bit 5 <-> STM Status/Status/Moving negative
//     Drive/Inputs/In/nState1 @bit 4 <-> STM Status/Status/Moving positive
//     Drive/Inputs/In/nState1 @bit 1 <-> STM Status/Status/Ready
//     Drive/Inputs/In/nState1 <-> STM Status/Status/Ready to enable
//     Drive/Inputs/In/nState1 @bit 6 <-> STM Status/Status/Torque reduced
//     Drive/Inputs/In/nState1 @bit 2 <-> STM Status/Status/Warning
//     Drive/Inputs/In/nState2 @bit 3 <-> STM Status/Status/Digital input 1
//     Drive/Inputs/In/nState2 @bit 4 <-> STM Status/Status/Digital input 2
//     Drive/Inputs/In/nState2 @bit 5 <-> STM Status/Status/Sync error
//     Drive/Inputs/In/nState2 @bit 7 <-> STM Status/Status/TxPDO Toggle
//     Drive/Inputs/In/nState4 @bit 1 <-> WcState/InputToggle
//     Drive/Inputs/In/nState4 <-> WcState/WcState
//     Drive/Outputs/Out/nCtrl1 <-> STM Control/Control/Enable
//     Drive/Outputs/Out/nCtrl1 @bit 2 <-> STM Control/Control/Reduce torque
//     Drive/Outputs/Out/nCtrl1 @bit 1 <-> STM Control/Control/Reset
//     Drive/Outputs/Out/nDataOut2[0] <-> STM Velocity/Velocity
//     Enc/Inputs/In/nDataIn1[0] <-> ENC Status compact/Counter value
//     Enc/Inputs/In/nDataIn2[0] <-> ENC Status compact/Latch value
//     Enc/Inputs/In/nState1 @bit 4 <-> ENC Status compact/Status/Counter overflow
//     Enc/Inputs/In/nState1 @bit 3 <-> ENC Status compact/Status/Counter underflow
//     Enc/Inputs/In/nState1 @bit 7 <-> ENC Status compact/Status/Extrapolation stall
//     Enc/Inputs/In/nState1 <-> ENC Status compact/Status/Latch C valid
//     Enc/Inputs/In/nState1 @bit 1 <-> ENC Status compact/Status/Latch extern valid
//     Enc/Inputs/In/nState1 @bit 2 <-> ENC Status compact/Status/Set counter done
//     Enc/Inputs/In/nState2 @bit 4 <-> ENC Status compact/Status/Status of extern latch
//     Enc/Inputs/In/nState2 <-> ENC Status compact/Status/Status of input A
//     Enc/Inputs/In/nState2 @bit 1 <-> ENC Status compact/Status/Status of input B
//     Enc/Inputs/In/nState2 @bit 2 <-> ENC Status compact/Status/Status of input C
//     Enc/Inputs/In/nState2 @bit 5 <-> ENC Status compact/Status/Sync error
//     Enc/Inputs/In/nState2 @bit 7 <-> ENC Status compact/Status/TxPDO Toggle
//     Enc/Inputs/In/nState4 @bit 1 <-> WcState/InputToggle
//     Enc/Inputs/In/nState4 <-> WcState/WcState
//     Enc/Outputs/Out/nCtrl1 <-> ENC Control compact/Control/Enable latch C
//     Enc/Outputs/Out/nCtrl1 @bit 3 <-> ENC Control compact/Control/Enable latch extern on negative edge
//     Enc/Outputs/Out/nCtrl1 @bit 1 <-> ENC Control compact/Control/Enable latch extern on positive edge
//     Enc/Outputs/Out/nCtrl1 @bit 2 <-> ENC Control compact/Control/Set counter
//     Enc/Outputs/Out/nDataOut1[0] <-> ENC Control compact/Set counter value
//   (this object) <-> Device 1 (EtherCAT)/Power (EK1200)/PLC Junction 2 (EK1122)/PLC Coupler 2 (EK1100)/PLC Junction 9 (EK1122)/SP1K4 Top Rail (EK1100)/SP1K4-EL5042-E7
//     Enc/Inputs/In/nComState @bit 1 <-> WcState/InputToggle
//     Enc/Inputs/In/nComState <-> WcState/WcState
//     Enc/Inputs/In/nDataIn1 <-> FB Inputs Channel 2/Position
//     Enc/Inputs/In/nDataIn1 <-> FB Inputs Channel 1/Position
//     Enc/Inputs/In/nState1 @bit 12 <-> FB Inputs Channel 2/Status/Diag
//     Enc/Inputs/In/nState1 @bit 12 <-> FB Inputs Channel 1/Status/Diag
//     Enc/Inputs/In/nState1 @bit 1 <-> FB Inputs Channel 2/Status/Error
//     Enc/Inputs/In/nState1 @bit 1 <-> FB Inputs Channel 1/Status/Error
//     Enc/Inputs/In/nState1 @bit 14 <-> FB Inputs Channel 2/Status/Input cycle counter
//     Enc/Inputs/In/nState1 @bit 14 <-> FB Inputs Channel 1/Status/Input cycle counter
//     Enc/Inputs/In/nState1 @bit 2 <-> FB Inputs Channel 2/Status/Ready
//     Enc/Inputs/In/nState1 @bit 2 <-> FB Inputs Channel 1/Status/Ready
//     Enc/Inputs/In/nState1 @bit 13 <-> FB Inputs Channel 2/Status/TxPDO State
//     Enc/Inputs/In/nState1 @bit 13 <-> FB Inputs Channel 1/Status/TxPDO State
//     Enc/Inputs/In/nState1 <-> FB Inputs Channel 2/Status/Warning
//     Enc/Inputs/In/nState1 <-> FB Inputs Channel 1/Status/Warning
//   (this object) <-> Device 1 (EtherCAT)/Power (EK1200)/PLC Junction 2 (EK1122)/PLC Coupler 2 (EK1100)/PLC Junction 9 (EK1122)/SP1K4 Top Rail (EK1100)/Thorlab-LenX-EL7031
//     Drive/Inputs/In/nState1 @bit 3 <-> STM Status/Status/Error
//     Drive/Inputs/In/nState1 @bit 5 <-> STM Status/Status/Moving negative
//     Drive/Inputs/In/nState1 @bit 4 <-> STM Status/Status/Moving positive
//     Drive/Inputs/In/nState1 @bit 1 <-> STM Status/Status/Ready
//     Drive/Inputs/In/nState1 <-> STM Status/Status/Ready to enable
//     Drive/Inputs/In/nState1 @bit 6 <-> STM Status/Status/Torque reduced
//     Drive/Inputs/In/nState1 @bit 2 <-> STM Status/Status/Warning
//     Drive/Inputs/In/nState2 @bit 3 <-> STM Status/Status/Digital input 1
//     Drive/Inputs/In/nState2 @bit 4 <-> STM Status/Status/Digital input 2
//     Drive/Inputs/In/nState2 @bit 5 <-> STM Status/Status/Sync error
//     Drive/Inputs/In/nState2 @bit 7 <-> STM Status/Status/TxPDO Toggle
//     Drive/Inputs/In/nState4 @bit 1 <-> WcState/InputToggle
//     Drive/Inputs/In/nState4 <-> WcState/WcState
//     Drive/Outputs/Out/nCtrl1 <-> STM Control/Control/Enable
//     Drive/Outputs/Out/nCtrl1 @bit 2 <-> STM Control/Control/Reduce torque
//     Drive/Outputs/Out/nCtrl1 @bit 1 <-> STM Control/Control/Reset
//     Drive/Outputs/Out/nDataOut2[0] <-> STM Velocity/Velocity
//   (this object) <-> Device 1 (EtherCAT)/Power (EK1200)/PLC Junction 2 (EK1122)/PLC Coupler 2 (EK1100)/PLC Junction 9 (EK1122)/SP1K4 Top Rail (EK1100)/FoilY-EL7041
//     Drive/Inputs/In/nState1 @bit 3 <-> STM Status/Status/Error
//     Drive/Inputs/In/nState1 @bit 5 <-> STM Status/Status/Moving negative
//     Drive/Inputs/In/nState1 @bit 4 <-> STM Status/Status/Moving positive
//     Drive/Inputs/In/nState1 @bit 1 <-> STM Status/Status/Ready
//     Drive/Inputs/In/nState1 <-> STM Status/Status/Ready to enable
//     Drive/Inputs/In/nState1 @bit 6 <-> STM Status/Status/Torque reduced
//     Drive/Inputs/In/nState1 @bit 2 <-> STM Status/Status/Warning
//     Drive/Inputs/In/nState2 @bit 3 <-> STM Status/Status/Digital input 1
//     Drive/Inputs/In/nState2 @bit 4 <-> STM Status/Status/Digital input 2
//     Drive/Inputs/In/nState2 @bit 5 <-> STM Status/Status/Sync error
//     Drive/Inputs/In/nState2 @bit 7 <-> STM Status/Status/TxPDO Toggle
//     Drive/Inputs/In/nState4 @bit 1 <-> WcState/InputToggle
//     Drive/Inputs/In/nState4 <-> WcState/WcState
//     Drive/Outputs/Out/nCtrl1 <-> STM Control/Control/Enable
//     Drive/Outputs/Out/nCtrl1 @bit 2 <-> STM Control/Control/Reduce torque
//     Drive/Outputs/Out/nCtrl1 @bit 1 <-> STM Control/Control/Reset
//     Drive/Outputs/Out/nDataOut2[0] <-> STM Velocity/Velocity
//   (this object) <-> Device 1 (EtherCAT)/Power (EK1200)/PLC Junction 2 (EK1122)/PLC Coupler 2 (EK1100)/PLC Junction 9 (EK1122)/LI2K4-PA1K4 (EK1100)/LI2K4-EL5042-E2
//     Enc/Inputs/In/nComState @bit 1 <-> WcState/InputToggle
//     Enc/Inputs/In/nComState <-> WcState/WcState
//     Enc/Inputs/In/nDataIn1 <-> FB Inputs Channel 1/Position
//     Enc/Inputs/In/nDataIn1 <-> FB Inputs Channel 2/Position
//     Enc/Inputs/In/nState1 @bit 12 <-> FB Inputs Channel 1/Status/Diag
//     Enc/Inputs/In/nState1 @bit 12 <-> FB Inputs Channel 2/Status/Diag
//     Enc/Inputs/In/nState1 @bit 1 <-> FB Inputs Channel 1/Status/Error
//     Enc/Inputs/In/nState1 @bit 1 <-> FB Inputs Channel 2/Status/Error
//     Enc/Inputs/In/nState1 @bit 14 <-> FB Inputs Channel 1/Status/Input cycle counter
//     Enc/Inputs/In/nState1 @bit 14 <-> FB Inputs Channel 2/Status/Input cycle counter
//     Enc/Inputs/In/nState1 @bit 2 <-> FB Inputs Channel 1/Status/Ready
//     Enc/Inputs/In/nState1 @bit 2 <-> FB Inputs Channel 2/Status/Ready
//     Enc/Inputs/In/nState1 @bit 13 <-> FB Inputs Channel 1/Status/TxPDO State
//     Enc/Inputs/In/nState1 @bit 13 <-> FB Inputs Channel 2/Status/TxPDO State
//     Enc/Inputs/In/nState1 <-> FB Inputs Channel 1/Status/Warning
//     Enc/Inputs/In/nState1 <-> FB Inputs Channel 2/Status/Warning
//   (this object) <-> Device 1 (EtherCAT)/Power (EK1200)/PLC Junction 2 (EK1122)/PLC Coupler 2 (EK1100)/PLC Junction 9 (EK1122)/LI2K4-PA1K4 (EK1100)/LI2K4Y-EL7047-E1
//     Drive/Inputs/In/nState1 @bit 3 <-> STM Status/Status/Error
//     Drive/Inputs/In/nState1 @bit 7 <-> STM Status/Status/Motor stall
//     Drive/Inputs/In/nState1 @bit 5 <-> STM Status/Status/Moving negative
//     Drive/Inputs/In/nState1 @bit 4 <-> STM Status/Status/Moving positive
//     Drive/Inputs/In/nState1 @bit 1 <-> STM Status/Status/Ready
//     Drive/Inputs/In/nState1 <-> STM Status/Status/Ready to enable
//     Drive/Inputs/In/nState1 @bit 6 <-> STM Status/Status/Torque reduced
//     Drive/Inputs/In/nState1 @bit 2 <-> STM Status/Status/Warning
//     Drive/Inputs/In/nState2 @bit 3 <-> STM Status/Status/Digital input 1
//     Drive/Inputs/In/nState2 @bit 4 <-> STM Status/Status/Digital input 2
//     Drive/Inputs/In/nState2 @bit 5 <-> STM Status/Status/Sync error
//     Drive/Inputs/In/nState2 @bit 7 <-> STM Status/Status/TxPDO Toggle
//     Drive/Inputs/In/nState4 @bit 1 <-> WcState/InputToggle
//     Drive/Inputs/In/nState4 <-> WcState/WcState
//     Drive/Outputs/Out/nCtrl1 <-> STM Control/Control/Enable
//     Drive/Outputs/Out/nCtrl1 @bit 2 <-> STM Control/Control/Reduce torque
//     Drive/Outputs/Out/nCtrl1 @bit 1 <-> STM Control/Control/Reset
//     Drive/Outputs/Out/nCtrl2 @bit 3 <-> STM Control/Control/Digital output 1
//     Drive/Outputs/Out/nDataOut2[0] <-> STM Velocity/Velocity
//   (this object) <-> Device 1 (EtherCAT)/Power (EK1200)/PLC Junction 2 (EK1122)/PLC Coupler 2 (EK1100)/PLC Junction 9 (EK1122)/LI2K4-PA1K4 (EK1100)/LI2K4X-EL7047-E3
//     Drive/Inputs/In/nState1 @bit 3 <-> STM Status/Status/Error
//     Drive/Inputs/In/nState1 @bit 7 <-> STM Status/Status/Motor stall
//     Drive/Inputs/In/nState1 @bit 5 <-> STM Status/Status/Moving negative
//     Drive/Inputs/In/nState1 @bit 4 <-> STM Status/Status/Moving positive
//     Drive/Inputs/In/nState1 @bit 1 <-> STM Status/Status/Ready
//     Drive/Inputs/In/nState1 <-> STM Status/Status/Ready to enable
//     Drive/Inputs/In/nState1 @bit 6 <-> STM Status/Status/Torque reduced
//     Drive/Inputs/In/nState1 @bit 2 <-> STM Status/Status/Warning
//     Drive/Inputs/In/nState2 @bit 3 <-> STM Status/Status/Digital input 1
//     Drive/Inputs/In/nState2 @bit 4 <-> STM Status/Status/Digital input 2
//     Drive/Inputs/In/nState2 @bit 5 <-> STM Status/Status/Sync error
//     Drive/Inputs/In/nState2 @bit 7 <-> STM Status/Status/TxPDO Toggle
//     Drive/Inputs/In/nState4 @bit 1 <-> WcState/InputToggle
//     Drive/Inputs/In/nState4 <-> WcState/WcState
//     Drive/Outputs/Out/nCtrl1 <-> STM Control/Control/Enable
//     Drive/Outputs/Out/nCtrl1 @bit 2 <-> STM Control/Control/Reduce torque
//     Drive/Outputs/Out/nCtrl1 @bit 1 <-> STM Control/Control/Reset
//     Drive/Outputs/Out/nCtrl2 @bit 3 <-> STM Control/Control/Digital output 1
//     Drive/Outputs/Out/nDataOut2[0] <-> STM Velocity/Velocity
//   (this object) <-> Device 1 (EtherCAT)/Power (EK1200)/PLC Junction 2 (EK1122)/PLC Coupler 2 (EK1100)/PLC Junction 9 (EK1122)/LI2K4-PA1K4 (EK1100)/PA1K4-PF-EL5042-E5
//     Enc/Inputs/In/nComState @bit 1 <-> WcState/InputToggle
//     Enc/Inputs/In/nComState <-> WcState/WcState
//     Enc/Inputs/In/nDataIn1 <-> FB Inputs Channel 1/Position
//     Enc/Inputs/In/nState1 @bit 12 <-> FB Inputs Channel 1/Status/Diag
//     Enc/Inputs/In/nState1 @bit 1 <-> FB Inputs Channel 1/Status/Error
//     Enc/Inputs/In/nState1 @bit 14 <-> FB Inputs Channel 1/Status/Input cycle counter
//     Enc/Inputs/In/nState1 @bit 2 <-> FB Inputs Channel 1/Status/Ready
//     Enc/Inputs/In/nState1 @bit 13 <-> FB Inputs Channel 1/Status/TxPDO State
//     Enc/Inputs/In/nState1 <-> FB Inputs Channel 1/Status/Warning
//   (this object) <-> Device 1 (EtherCAT)/Power (EK1200)/PLC Junction 2 (EK1122)/PLC Coupler 2 (EK1100)/PLC Junction 9 (EK1122)/LI2K4-PA1K4 (EK1100)/PA1K4-PF-EL7047-E4
//     Drive/Inputs/In/nState1 @bit 3 <-> STM Status/Status/Error
//     Drive/Inputs/In/nState1 @bit 7 <-> STM Status/Status/Motor stall
//     Drive/Inputs/In/nState1 @bit 5 <-> STM Status/Status/Moving negative
//     Drive/Inputs/In/nState1 @bit 4 <-> STM Status/Status/Moving positive
//     Drive/Inputs/In/nState1 @bit 1 <-> STM Status/Status/Ready
//     Drive/Inputs/In/nState1 <-> STM Status/Status/Ready to enable
//     Drive/Inputs/In/nState1 @bit 6 <-> STM Status/Status/Torque reduced
//     Drive/Inputs/In/nState1 @bit 2 <-> STM Status/Status/Warning
//     Drive/Inputs/In/nState2 @bit 3 <-> STM Status/Status/Digital input 1
//     Drive/Inputs/In/nState2 @bit 4 <-> STM Status/Status/Digital input 2
//     Drive/Inputs/In/nState2 @bit 5 <-> STM Status/Status/Sync error
//     Drive/Inputs/In/nState2 @bit 7 <-> STM Status/Status/TxPDO Toggle
//     Drive/Inputs/In/nState4 @bit 1 <-> WcState/InputToggle
//     Drive/Inputs/In/nState4 <-> WcState/WcState
//     Drive/Outputs/Out/nCtrl1 <-> STM Control/Control/Enable
//     Drive/Outputs/Out/nCtrl1 @bit 2 <-> STM Control/Control/Reduce torque
//     Drive/Outputs/Out/nCtrl1 @bit 1 <-> STM Control/Control/Reset
//     Drive/Outputs/Out/nCtrl2 @bit 3 <-> STM Control/Control/Digital output 1
//     Drive/Outputs/Out/nDataOut2[0] <-> STM Velocity/Velocity
//   tmo_motion Instance <-> Device 1 (EtherCAT)/Power (EK1200)/PLC Junction 1 (EK1122)/X2 TMO FEE EC2 (EK1100)/FEE EC2 E1 (EK1122)/X1 AL1K4-L2SI (EK1100)/AL1K4-EL2004-E3
//     PlcTask Outputs/Main.M1.bBrakeRelease <-> Channel 1/Output
//   tmo_motion Instance <-> Device 1 (EtherCAT)/Power (EK1200)/PLC Junction 1 (EK1122)/X2 TMO FEE EC2 (EK1100)/FEE EC2 E1 (EK1122)/X1 AL1K4-L2SI (EK1100)/AL1K4-EL4004-E4
//     PlcTask Outputs/PRG_AL1K4_L2SI.fbAL1K4.fbLaser.iLaserINT <-> AO Outputs Channel 1/Analog output
//     PlcTask Outputs/PRG_AL1K4_L2SI.fbAL1K4.fbLaser.iShutdownINT <-> AO Outputs Channel 2/Analog output
//   tmo_motion Instance <-> Device 1 (EtherCAT)/Power (EK1200)/PLC Junction 1 (EK1122)/X2 TMO FEE EC2 (EK1100)/FEE EC2 E1 (EK1122)/X1 AL1K4-L2SI (EK1100)/AL1K4-EL5042-E2
//     PlcTask Inputs/Main.M1.nRawEncoderULINT <-> FB Inputs Channel 1/Position
//   tmo_motion Instance <-> Device 1 (EtherCAT)/Power (EK1200)/PLC Junction 1 (EK1122)/X2 TMO FEE EC2 (EK1100)/FEE EC2 E1 (EK1122)/X1 AL1K4-L2SI (EK1100)/AL1K4-EL7041-E1
//     PlcTask Inputs/Main.M1.bLimitBackwardEnable <-> STM Status/Status/Digital input 2
//     PlcTask Inputs/Main.M1.bLimitForwardEnable <-> STM Status/Status/Digital input 1
//   tmo_motion Instance <-> Device 1 (EtherCAT)/Power (EK1200)/PLC Junction 1 (EK1122)/X2 TMO FEE EC2 (EK1100)/FEE EC2 E1 (EK1122)/X2 SL1K4-SCATTER/SL1K4-EL5101-E2
//     PlcTask Inputs/Main.M10.nRawEncoderUINT <-> ENC Status compact/Counter value
//   tmo_motion Instance <-> Device 1 (EtherCAT)/Power (EK1200)/PLC Junction 1 (EK1122)/X2 TMO FEE EC2 (EK1100)/FEE EC2 E1 (EK1122)/X2 SL1K4-SCATTER/SL1K4-EL5101-E4
//     PlcTask Inputs/Main.M11.nRawEncoderUINT <-> ENC Status compact/Counter value
//   tmo_motion Instance <-> Device 1 (EtherCAT)/Power (EK1200)/PLC Junction 1 (EK1122)/X2 TMO FEE EC2 (EK1100)/FEE EC2 E1 (EK1122)/X2 SL1K4-SCATTER/SL1K4-EL5101-E6
//     PlcTask Inputs/Main.M12.nRawEncoderUINT <-> ENC Status compact/Counter value
//   tmo_motion Instance <-> Device 1 (EtherCAT)/Power (EK1200)/PLC Junction 1 (EK1122)/X2 TMO FEE EC2 (EK1100)/FEE EC2 E1 (EK1122)/X2 SL1K4-SCATTER/SL1K4-EL5101-E8
//     PlcTask Inputs/Main.M13.nRawEncoderUINT <-> ENC Status compact/Counter value
//   tmo_motion Instance <-> Device 1 (EtherCAT)/Power (EK1200)/PLC Junction 1 (EK1122)/X2 TMO FEE EC2 (EK1100)/FEE EC2 E1 (EK1122)/X2 SL1K4-SCATTER/SL1K4-EL7031-E1
//     PlcTask Inputs/Main.M10.bLimitBackwardEnable <-> STM Status/Status/Digital input 1
//     PlcTask Inputs/Main.M10.bLimitForwardEnable <-> STM Status/Status/Digital input 2
//   tmo_motion Instance <-> Device 1 (EtherCAT)/Power (EK1200)/PLC Junction 1 (EK1122)/X2 TMO FEE EC2 (EK1100)/FEE EC2 E1 (EK1122)/X2 SL1K4-SCATTER/SL1K4-EL7031-E3
//     PlcTask Inputs/Main.M11.bLimitBackwardEnable <-> STM Status/Status/Digital input 1
//     PlcTask Inputs/Main.M11.bLimitForwardEnable <-> STM Status/Status/Digital input 2
//   tmo_motion Instance <-> Device 1 (EtherCAT)/Power (EK1200)/PLC Junction 1 (EK1122)/X2 TMO FEE EC2 (EK1100)/FEE EC2 E1 (EK1122)/X2 SL1K4-SCATTER/SL1K4-EL7031-E5
//     PlcTask Inputs/Main.M12.bLimitBackwardEnable <-> STM Status/Status/Digital input 2
//     PlcTask Inputs/Main.M12.bLimitForwardEnable <-> STM Status/Status/Digital input 1
//   tmo_motion Instance <-> Device 1 (EtherCAT)/Power (EK1200)/PLC Junction 1 (EK1122)/X2 TMO FEE EC2 (EK1100)/FEE EC2 E1 (EK1122)/X2 SL1K4-SCATTER/SL1K4-EL7031-E7
//     PlcTask Inputs/Main.M13.bLimitBackwardEnable <-> STM Status/Status/Digital input 2
//     PlcTask Inputs/Main.M13.bLimitForwardEnable <-> STM Status/Status/Digital input 1
//   tmo_motion Instance <-> Device 1 (EtherCAT)/Power (EK1200)/PLC Junction 1 (EK1122)/X2 TMO FEE EC2 (EK1100)/FEE EC2 E2 (EK1122)/X1 IM2K4-PPM (EK1100)/IM2K4-EL1004-E8
//     PlcTask Inputs/PRG_IM2K4_PPM.fbIM2K4.fbFlowSwitch.bFlowOk <-> Channel 1/Input
//   tmo_motion Instance <-> Device 1 (EtherCAT)/Power (EK1200)/PLC Junction 1 (EK1122)/X2 TMO FEE EC2 (EK1100)/FEE EC2 E2 (EK1122)/X1 IM2K4-PPM (EK1100)/IM2K4-EL2004-E3
//     PlcTask Outputs/Main.M9.bBrakeRelease <-> Channel 1/Output
//     PlcTask Outputs/PRG_IM2K4_PPM.fbIM2K4.fbGige.bGigePower <-> Channel 2/Output
//   tmo_motion Instance <-> Device 1 (EtherCAT)/Power (EK1200)/PLC Junction 1 (EK1122)/X2 TMO FEE EC2 (EK1100)/FEE EC2 E2 (EK1122)/X1 IM2K4-PPM (EK1100)/IM2K4-EL3062-E6
//     PlcTask Inputs/PRG_IM2K4_PPM.fbIM2K4.fbPowerMeter.iVoltageINT <-> AI Standard Channel 1/Value
//   tmo_motion Instance <-> Device 1 (EtherCAT)/Power (EK1200)/PLC Junction 1 (EK1122)/X2 TMO FEE EC2 (EK1100)/FEE EC2 E2 (EK1122)/X1 IM2K4-PPM (EK1100)/IM2K4-EL3314-E4
//     PlcTask Inputs/PRG_IM2K4_PPM.fbIM2K4.fbPowerMeter.fbTempSensor.bError <-> TC Inputs Channel 1/Status/Error
//     PlcTask Inputs/PRG_IM2K4_PPM.fbIM2K4.fbPowerMeter.fbTempSensor.bOverrange <-> TC Inputs Channel 1/Status/Overrange
//     PlcTask Inputs/PRG_IM2K4_PPM.fbIM2K4.fbPowerMeter.fbTempSensor.bUnderrange <-> TC Inputs Channel 1/Status/Underrange
//     PlcTask Inputs/PRG_IM2K4_PPM.fbIM2K4.fbPowerMeter.fbTempSensor.iRaw <-> TC Inputs Channel 1/Value
//     PlcTask Inputs/PRG_IM2K4_PPM.fbIM2K4.fbYagTempSensor.bError <-> TC Inputs Channel 2/Status/Error
//     PlcTask Inputs/PRG_IM2K4_PPM.fbIM2K4.fbYagTempSensor.bOverrange <-> TC Inputs Channel 2/Status/Overrange
//     PlcTask Inputs/PRG_IM2K4_PPM.fbIM2K4.fbYagTempSensor.bUnderrange <-> TC Inputs Channel 2/Status/Underrange
//     PlcTask Inputs/PRG_IM2K4_PPM.fbIM2K4.fbYagTempSensor.iRaw <-> TC Inputs Channel 2/Value
//   tmo_motion Instance <-> Device 1 (EtherCAT)/Power (EK1200)/PLC Junction 1 (EK1122)/X2 TMO FEE EC2 (EK1100)/FEE EC2 E2 (EK1122)/X1 IM2K4-PPM (EK1100)/IM2K4-EL4004-E7
//     PlcTask Outputs/PRG_IM2K4_PPM.fbIM2K4.fbGige.iIlluminatorINT <-> AO Outputs Channel 1/Analog output
//   tmo_motion Instance <-> Device 1 (EtherCAT)/Power (EK1200)/PLC Junction 1 (EK1122)/X2 TMO FEE EC2 (EK1100)/FEE EC2 E2 (EK1122)/X1 IM2K4-PPM (EK1100)/IM2K4-EL5042-E2
//     PlcTask Inputs/Main.M9.nRawEncoderULINT <-> FB Inputs Channel 1/Position
//   tmo_motion Instance <-> Device 1 (EtherCAT)/Power (EK1200)/PLC Junction 1 (EK1122)/X2 TMO FEE EC2 (EK1100)/FEE EC2 E2 (EK1122)/X1 IM2K4-PPM (EK1100)/IM2K4-EL7041-E1
//     PlcTask Inputs/Main.M9.bLimitBackwardEnable <-> STM Status/Status/Digital input 2
//     PlcTask Inputs/Main.M9.bLimitForwardEnable <-> STM Status/Status/Digital input 1
//   tmo_motion Instance <-> Device 1 (EtherCAT)/Power (EK1200)/PLC Junction 2 (EK1122)/PLC Coupler 1(EK1100)/PLC Junction 5 (EK1122)/IM3K4-PPM (EK1100)/IM3K4-EL2004-E3
//     PlcTask Outputs/Main.M15.bBrakeRelease <-> Channel 1/Output
//     PlcTask Outputs/PRG_IM3K4_PPM.fbIM3K4.fbGige.bGigePower <-> Channel 2/Output
//   tmo_motion Instance <-> Device 1 (EtherCAT)/Power (EK1200)/PLC Junction 2 (EK1122)/PLC Coupler 1(EK1100)/PLC Junction 5 (EK1122)/IM3K4-PPM (EK1100)/IM3K4-EL3062-E6
//     PlcTask Inputs/PRG_IM3K4_PPM.fbIM3K4.fbPowerMeter.iVoltageINT <-> AI Standard Channel 1/Value
//   tmo_motion Instance <-> Device 1 (EtherCAT)/Power (EK1200)/PLC Junction 2 (EK1122)/PLC Coupler 1(EK1100)/PLC Junction 5 (EK1122)/IM3K4-PPM (EK1100)/IM3K4-EL3314-E4
//     PlcTask Inputs/PRG_IM3K4_PPM.fbIM3K4.fbPowerMeter.fbTempSensor.bError <-> TC Inputs Channel 1/Status/Error
//     PlcTask Inputs/PRG_IM3K4_PPM.fbIM3K4.fbPowerMeter.fbTempSensor.bOverrange <-> TC Inputs Channel 1/Status/Overrange
//     PlcTask Inputs/PRG_IM3K4_PPM.fbIM3K4.fbPowerMeter.fbTempSensor.bUnderrange <-> TC Inputs Channel 1/Status/Underrange
//     PlcTask Inputs/PRG_IM3K4_PPM.fbIM3K4.fbPowerMeter.fbTempSensor.iRaw <-> TC Inputs Channel 1/Value
//     PlcTask Inputs/PRG_IM3K4_PPM.fbIM3K4.fbYagTempSensor.bError <-> TC Inputs Channel 2/Status/Error
//     PlcTask Inputs/PRG_IM3K4_PPM.fbIM3K4.fbYagTempSensor.bOverrange <-> TC Inputs Channel 2/Status/Overrange
//     PlcTask Inputs/PRG_IM3K4_PPM.fbIM3K4.fbYagTempSensor.bUnderrange <-> TC Inputs Channel 2/Status/Underrange
//     PlcTask Inputs/PRG_IM3K4_PPM.fbIM3K4.fbYagTempSensor.iRaw <-> TC Inputs Channel 2/Value
//   tmo_motion Instance <-> Device 1 (EtherCAT)/Power (EK1200)/PLC Junction 2 (EK1122)/PLC Coupler 1(EK1100)/PLC Junction 5 (EK1122)/IM3K4-PPM (EK1100)/IM3K4-EL4004-E7
//     PlcTask Outputs/PRG_IM3K4_PPM.fbIM3K4.fbGige.iIlluminatorINT <-> AO Outputs Channel 1/Analog output
//   tmo_motion Instance <-> Device 1 (EtherCAT)/Power (EK1200)/PLC Junction 2 (EK1122)/PLC Coupler 1(EK1100)/PLC Junction 5 (EK1122)/IM3K4-PPM (EK1100)/IM3K4-EL5042-E2
//     PlcTask Inputs/Main.M15.nRawEncoderULINT <-> FB Inputs Channel 1/Position
//   tmo_motion Instance <-> Device 1 (EtherCAT)/Power (EK1200)/PLC Junction 2 (EK1122)/PLC Coupler 1(EK1100)/PLC Junction 5 (EK1122)/IM3K4-PPM (EK1100)/IM3K4-EL7041-E1
//     PlcTask Inputs/Main.M15.bLimitBackwardEnable <-> STM Status/Status/Digital input 2
//     PlcTask Inputs/Main.M15.bLimitForwardEnable <-> STM Status/Status/Digital input 1
//   tmo_motion Instance <-> Device 1 (EtherCAT)/Power (EK1200)/PLC Junction 2 (EK1122)/PLC Coupler 1(EK1100)/PLC Junction 5 (EK1122)/IM4K4-PPM (EK1100)/IM4K4-EL2004-E3
//     PlcTask Outputs/Main.M16.bBrakeRelease <-> Channel 1/Output
//     PlcTask Outputs/PRG_IM4K4_PPM.fbIM4K4.fbGige.bGigePower <-> Channel 2/Output
//   tmo_motion Instance <-> Device 1 (EtherCAT)/Power (EK1200)/PLC Junction 2 (EK1122)/PLC Coupler 1(EK1100)/PLC Junction 5 (EK1122)/IM4K4-PPM (EK1100)/IM4K4-EL3052-E5
//     PlcTask Inputs/PRG_IM3K4_PPM.fbIM3K4.fbFlowMeter.iRaw <-> AI Standard Channel 1/Value
//     PlcTask Inputs/PRG_IM4K4_PPM.fbIM4K4.fbFlowMeter.iRaw <-> AI Standard Channel 1/Value
//   tmo_motion Instance <-> Device 1 (EtherCAT)/Power (EK1200)/PLC Junction 2 (EK1122)/PLC Coupler 1(EK1100)/PLC Junction 5 (EK1122)/IM4K4-PPM (EK1100)/IM4K4-EL3062-E6
//     PlcTask Inputs/PRG_IM4K4_PPM.fbIM4K4.fbPowerMeter.iVoltageINT <-> AI Standard Channel 1/Value
//   tmo_motion Instance <-> Device 1 (EtherCAT)/Power (EK1200)/PLC Junction 2 (EK1122)/PLC Coupler 1(EK1100)/PLC Junction 5 (EK1122)/IM4K4-PPM (EK1100)/IM4K4-EL3314-E4
//     PlcTask Inputs/PRG_IM4K4_PPM.fbIM4K4.fbPowerMeter.fbTempSensor.bError <-> TC Inputs Channel 1/Status/Error
//     PlcTask Inputs/PRG_IM4K4_PPM.fbIM4K4.fbPowerMeter.fbTempSensor.bOverrange <-> TC Inputs Channel 1/Status/Overrange
//     PlcTask Inputs/PRG_IM4K4_PPM.fbIM4K4.fbPowerMeter.fbTempSensor.bUnderrange <-> TC Inputs Channel 1/Status/Underrange
//     PlcTask Inputs/PRG_IM4K4_PPM.fbIM4K4.fbPowerMeter.fbTempSensor.iRaw <-> TC Inputs Channel 1/Value
//     PlcTask Inputs/PRG_IM4K4_PPM.fbIM4K4.fbYagTempSensor.bError <-> TC Inputs Channel 2/Status/Error
//     PlcTask Inputs/PRG_IM4K4_PPM.fbIM4K4.fbYagTempSensor.bOverrange <-> TC Inputs Channel 2/Status/Overrange
//     PlcTask Inputs/PRG_IM4K4_PPM.fbIM4K4.fbYagTempSensor.bUnderrange <-> TC Inputs Channel 2/Status/Underrange
//     PlcTask Inputs/PRG_IM4K4_PPM.fbIM4K4.fbYagTempSensor.iRaw <-> TC Inputs Channel 2/Value
//   tmo_motion Instance <-> Device 1 (EtherCAT)/Power (EK1200)/PLC Junction 2 (EK1122)/PLC Coupler 1(EK1100)/PLC Junction 5 (EK1122)/IM4K4-PPM (EK1100)/IM4K4-EL4004-E7
//     PlcTask Outputs/PRG_IM4K4_PPM.fbIM4K4.fbGige.iIlluminatorINT <-> AO Outputs Channel 1/Analog output
//   tmo_motion Instance <-> Device 1 (EtherCAT)/Power (EK1200)/PLC Junction 2 (EK1122)/PLC Coupler 1(EK1100)/PLC Junction 5 (EK1122)/IM4K4-PPM (EK1100)/IM4K4-EL5042-E2
//     PlcTask Inputs/Main.M16.nRawEncoderULINT <-> FB Inputs Channel 1/Position
//   tmo_motion Instance <-> Device 1 (EtherCAT)/Power (EK1200)/PLC Junction 2 (EK1122)/PLC Coupler 1(EK1100)/PLC Junction 5 (EK1122)/IM4K4-PPM (EK1100)/IM4K4-EL7041-E1
//     PlcTask Inputs/Main.M16.bLimitBackwardEnable <-> STM Status/Status/Digital input 2
//     PlcTask Inputs/Main.M16.bLimitForwardEnable <-> STM Status/Status/Digital input 1
//   tmo_motion Instance <-> Device 1 (EtherCAT)/Power (EK1200)/PLC Junction 2 (EK1122)/PLC Coupler 1(EK1100)/PLC Junction 6 (EK1122)/LI1K4-LIC (EK1100)/LI1K4-EL2004-E3
//     PlcTask Outputs/Main.M20.bBrakeRelease <-> Channel 1/Output
//   tmo_motion Instance <-> Device 1 (EtherCAT)/Power (EK1200)/PLC Junction 2 (EK1122)/PLC Coupler 1(EK1100)/PLC Junction 6 (EK1122)/LI1K4-LIC (EK1100)/LI1K4-EL5042-E2
//     PlcTask Inputs/Main.M20.nRawEncoderULINT <-> FB Inputs Channel 1/Position
//   tmo_motion Instance <-> Device 1 (EtherCAT)/Power (EK1200)/PLC Junction 2 (EK1122)/PLC Coupler 1(EK1100)/PLC Junction 6 (EK1122)/LI1K4-LIC (EK1100)/LI1K4-EL7041-E1
//     PlcTask Inputs/Main.M20.bLimitBackwardEnable <-> STM Status/Status/Digital input 2
//     PlcTask Inputs/Main.M20.bLimitForwardEnable <-> STM Status/Status/Digital input 1
//   tmo_motion Instance <-> Device 1 (EtherCAT)/Power (EK1200)/PLC Junction 2 (EK1122)/PLC Coupler 2 (EK1100)/PLC Junction 10 (EK1122)/Granite3 (EK1100)/PLC Junction 11 (EK1122)/PF2K4-WFS (EK1100)/PF2K4-EL2004-E4
//     PlcTask Outputs/Main.M28.bBrakeRelease <-> Channel 1/Output
//   tmo_motion Instance <-> Device 1 (EtherCAT)/Power (EK1200)/PLC Junction 2 (EK1122)/PLC Coupler 2 (EK1100)/PLC Junction 10 (EK1122)/Granite3 (EK1100)/PLC Junction 11 (EK1122)/PF2K4-WFS (EK1100)/PF2K4-EL3314-E5
//     PlcTask Inputs/PRG_PF2K4_WFS_TARGET.fbPF2K4.fbThermoCouple1.bError <-> TC Inputs Channel 1/Status/Error
//     PlcTask Inputs/PRG_PF2K4_WFS_TARGET.fbPF2K4.fbThermoCouple2.bError <-> TC Inputs Channel 2/Status/Error
//     PlcTask Inputs/PRG_PF2K4_WFS_TARGET.fbPF2K4.fbThermoCouple1.bOverrange <-> TC Inputs Channel 1/Status/Overrange
//     PlcTask Inputs/PRG_PF2K4_WFS_TARGET.fbPF2K4.fbThermoCouple2.bOverrange <-> TC Inputs Channel 2/Status/Overrange
//     PlcTask Inputs/PRG_PF2K4_WFS_TARGET.fbPF2K4.fbThermoCouple1.bUnderrange <-> TC Inputs Channel 1/Status/Underrange
//     PlcTask Inputs/PRG_PF2K4_WFS_TARGET.fbPF2K4.fbThermoCouple2.bUnderrange <-> TC Inputs Channel 2/Status/Underrange
//     PlcTask Inputs/PRG_PF2K4_WFS_TARGET.fbPF2K4.fbThermoCouple1.iRaw <-> TC Inputs Channel 1/Value
//     PlcTask Inputs/PRG_PF2K4_WFS_TARGET.fbPF2K4.fbThermoCouple2.iRaw <-> TC Inputs Channel 2/Value
//   tmo_motion Instance <-> Device 1 (EtherCAT)/Power (EK1200)/PLC Junction 2 (EK1122)/PLC Coupler 2 (EK1100)/PLC Junction 10 (EK1122)/Granite3 (EK1100)/PLC Junction 11 (EK1122)/PF2K4-WFS (EK1100)/PF2K4-EL5042-E3
//     PlcTask Inputs/Main.M28.nRawEncoderULINT <-> FB Inputs Channel 2/Position
//     PlcTask Inputs/Main.M29.nRawEncoderULINT <-> FB Inputs Channel 1/Position
//   tmo_motion Instance <-> Device 1 (EtherCAT)/Power (EK1200)/PLC Junction 2 (EK1122)/PLC Coupler 2 (EK1100)/PLC Junction 10 (EK1122)/Granite3 (EK1100)/PLC Junction 11 (EK1122)/PF2K4-WFS (EK1100)/PF2K4-EL7041-E1
//     PlcTask Inputs/Main.M28.bLimitBackwardEnable <-> STM Status/Status/Digital input 2
//     PlcTask Inputs/Main.M28.bLimitForwardEnable <-> STM Status/Status/Digital input 1
//   tmo_motion Instance <-> Device 1 (EtherCAT)/Power (EK1200)/PLC Junction 2 (EK1122)/PLC Coupler 2 (EK1100)/PLC Junction 10 (EK1122)/Granite3 (EK1100)/PLC Junction 12  (EK1122)/IM6K4 (EK1100)/IM6K4-EL2004-E3
//     PlcTask Outputs/Main.M27.bBrakeRelease <-> Channel 1/Output
//     PlcTask Outputs/PRG_IM6K4_PPM.fbIM6K4.fbGige.bGigePower <-> Channel 2/Output
//   tmo_motion Instance <-> Device 1 (EtherCAT)/Power (EK1200)/PLC Junction 2 (EK1122)/PLC Coupler 2 (EK1100)/PLC Junction 10 (EK1122)/Granite3 (EK1100)/PLC Junction 12  (EK1122)/IM6K4 (EK1100)/IM6K4-EL3052-E5
//     PlcTask Inputs/PRG_IM6K4_PPM.fbIM6K4.fbFlowMeter.iRaw <-> AI Standard Channel 1/Value
//     PlcTask Inputs/PRG_PF2K4_WFS_TARGET.fbPF2K4.fbFlowMeter.iRaw <-> AI Standard Channel 1/Value
//     PlcTask Inputs/PRG_TM2K4.fbTM2K4.fbFlowMeter.iRaw <-> AI Standard Channel 1/Value
//   tmo_motion Instance <-> Device 1 (EtherCAT)/Power (EK1200)/PLC Junction 2 (EK1122)/PLC Coupler 2 (EK1100)/PLC Junction 10 (EK1122)/Granite3 (EK1100)/PLC Junction 12  (EK1122)/IM6K4 (EK1100)/IM6K4-EL3062-E6
//     PlcTask Inputs/PRG_IM6K4_PPM.fbIM6K4.fbPowerMeter.iVoltageINT <-> AI Standard Channel 1/Value
//   tmo_motion Instance <-> Device 1 (EtherCAT)/Power (EK1200)/PLC Junction 2 (EK1122)/PLC Coupler 2 (EK1100)/PLC Junction 10 (EK1122)/Granite3 (EK1100)/PLC Junction 12  (EK1122)/IM6K4 (EK1100)/IM6K4-EL3314-E4
//     PlcTask Inputs/PRG_IM6K4_PPM.fbIM6K4.fbPowerMeter.fbTempSensor.bError <-> TC Inputs Channel 1/Status/Error
//     PlcTask Inputs/PRG_IM6K4_PPM.fbIM6K4.fbPowerMeter.fbTempSensor.bOverrange <-> TC Inputs Channel 1/Status/Overrange
//     PlcTask Inputs/PRG_IM6K4_PPM.fbIM6K4.fbPowerMeter.fbTempSensor.bUnderrange <-> TC Inputs Channel 1/Status/Underrange
//     PlcTask Inputs/PRG_IM6K4_PPM.fbIM6K4.fbPowerMeter.fbTempSensor.iRaw <-> TC Inputs Channel 1/Value
//     PlcTask Inputs/PRG_IM6K4_PPM.fbIM6K4.fbYagTempSensor.bError <-> TC Inputs Channel 2/Status/Error
//     PlcTask Inputs/PRG_IM6K4_PPM.fbIM6K4.fbYagTempSensor.bOverrange <-> TC Inputs Channel 2/Status/Overrange
//     PlcTask Inputs/PRG_IM6K4_PPM.fbIM6K4.fbYagTempSensor.bUnderrange <-> TC Inputs Channel 2/Status/Underrange
//     PlcTask Inputs/PRG_IM6K4_PPM.fbIM6K4.fbYagTempSensor.iRaw <-> TC Inputs Channel 2/Value
//   tmo_motion Instance <-> Device 1 (EtherCAT)/Power (EK1200)/PLC Junction 2 (EK1122)/PLC Coupler 2 (EK1100)/PLC Junction 10 (EK1122)/Granite3 (EK1100)/PLC Junction 12  (EK1122)/IM6K4 (EK1100)/IM6K4-EL4004-E7
//     PlcTask Outputs/PRG_IM6K4_PPM.fbIM6K4.fbGige.iIlluminatorINT <-> AO Outputs Channel 1/Analog output
//   tmo_motion Instance <-> Device 1 (EtherCAT)/Power (EK1200)/PLC Junction 2 (EK1122)/PLC Coupler 2 (EK1100)/PLC Junction 10 (EK1122)/Granite3 (EK1100)/PLC Junction 12  (EK1122)/IM6K4 (EK1100)/IM6K4-EL5042-E2
//     PlcTask Inputs/Main.M27.nRawEncoderULINT <-> FB Inputs Channel 1/Position
//   tmo_motion Instance <-> Device 1 (EtherCAT)/Power (EK1200)/PLC Junction 2 (EK1122)/PLC Coupler 2 (EK1100)/PLC Junction 10 (EK1122)/Granite3 (EK1100)/PLC Junction 12  (EK1122)/IM6K4 (EK1100)/IM6K4-EL7041-E1
//     PlcTask Inputs/Main.M27.bLimitBackwardEnable <-> STM Status/Status/Digital input 2
//     PlcTask Inputs/Main.M27.bLimitForwardEnable <-> STM Status/Status/Digital input 1
//   tmo_motion Instance <-> Device 1 (EtherCAT)/Power (EK1200)/PLC Junction 2 (EK1122)/PLC Coupler 2 (EK1100)/PLC Junction 10 (EK1122)/Granite3 (EK1100)/PLC Junction 12  (EK1122)/TM2K4 (EK1100)/TM2K4-EL2004-E4
//     PlcTask Outputs/Main.M30.bBrakeRelease <-> Channel 1/Output
//   tmo_motion Instance <-> Device 1 (EtherCAT)/Power (EK1200)/PLC Junction 2 (EK1122)/PLC Coupler 2 (EK1100)/PLC Junction 10 (EK1122)/Granite3 (EK1100)/PLC Junction 12  (EK1122)/TM2K4 (EK1100)/TM2K4-EL3314-E5
//     PlcTask Inputs/PRG_TM2K4.fbTM2K4.fbTempSensor1.bError <-> TC Inputs Channel 1/Status/Error
//     PlcTask Inputs/PRG_TM2K4.fbTM2K4.fbTempSensor1.bOverrange <-> TC Inputs Channel 1/Status/Overrange
//     PlcTask Inputs/PRG_TM2K4.fbTM2K4.fbTempSensor1.bUnderrange <-> TC Inputs Channel 1/Status/Underrange
//     PlcTask Inputs/PRG_TM2K4.fbTM2K4.fbTempSensor1.iRaw <-> TC Inputs Channel 1/Value
//   tmo_motion Instance <-> Device 1 (EtherCAT)/Power (EK1200)/PLC Junction 2 (EK1122)/PLC Coupler 2 (EK1100)/PLC Junction 10 (EK1122)/Granite3 (EK1100)/PLC Junction 12  (EK1122)/TM2K4 (EK1100)/TM2K4-EL5042-E3
//     PlcTask Inputs/Main.M30.nRawEncoderULINT <-> FB Inputs Channel 1/Position
//     PlcTask Inputs/Main.M31.nRawEncoderULINT <-> FB Inputs Channel 2/Position
//   tmo_motion Instance <-> Device 1 (EtherCAT)/Power (EK1200)/PLC Junction 2 (EK1122)/PLC Coupler 2 (EK1100)/PLC Junction 10 (EK1122)/Granite3 (EK1100)/PLC Junction 12  (EK1122)/TM2K4 (EK1100)/TM2K4-EL7041-E1
//     PlcTask Inputs/Main.M30.bLimitBackwardEnable <-> STM Status/Status/Digital input 2
//     PlcTask Inputs/Main.M30.bLimitForwardEnable <-> STM Status/Status/Digital input 1
//   tmo_motion Instance <-> Device 1 (EtherCAT)/Power (EK1200)/PLC Junction 2 (EK1122)/PLC Coupler 2 (EK1100)/PLC Junction 10 (EK1122)/PF1K4-WFS (EK1100)/PF1K4-EL2004-E4
//     PlcTask Outputs/Main.M18.bBrakeRelease <-> Channel 1/Output
//   tmo_motion Instance <-> Device 1 (EtherCAT)/Power (EK1200)/PLC Junction 2 (EK1122)/PLC Coupler 2 (EK1100)/PLC Junction 10 (EK1122)/PF1K4-WFS (EK1100)/PF1K4-EL3314-E5
//     PlcTask Inputs/PRG_PF1K4_WFS_TARGET.fbPF1K4.fbThermoCouple1.bError <-> TC Inputs Channel 1/Status/Error
//     PlcTask Inputs/PRG_PF1K4_WFS_TARGET.fbPF1K4.fbThermoCouple2.bError <-> TC Inputs Channel 2/Status/Error
//     PlcTask Inputs/PRG_PF1K4_WFS_TARGET.fbPF1K4.fbThermoCouple1.bOverrange <-> TC Inputs Channel 1/Status/Overrange
//     PlcTask Inputs/PRG_PF1K4_WFS_TARGET.fbPF1K4.fbThermoCouple2.bOverrange <-> TC Inputs Channel 2/Status/Overrange
//     PlcTask Inputs/PRG_PF1K4_WFS_TARGET.fbPF1K4.fbThermoCouple1.bUnderrange <-> TC Inputs Channel 1/Status/Underrange
//     PlcTask Inputs/PRG_PF1K4_WFS_TARGET.fbPF1K4.fbThermoCouple2.bUnderrange <-> TC Inputs Channel 2/Status/Underrange
//     PlcTask Inputs/PRG_PF1K4_WFS_TARGET.fbPF1K4.fbThermoCouple1.iRaw <-> TC Inputs Channel 1/Value
//     PlcTask Inputs/PRG_PF1K4_WFS_TARGET.fbPF1K4.fbThermoCouple2.iRaw <-> TC Inputs Channel 2/Value
//   tmo_motion Instance <-> Device 1 (EtherCAT)/Power (EK1200)/PLC Junction 2 (EK1122)/PLC Coupler 2 (EK1100)/PLC Junction 10 (EK1122)/PF1K4-WFS (EK1100)/PF1K4-EL5042-E3
//     PlcTask Inputs/Main.M18.nRawEncoderULINT <-> FB Inputs Channel 2/Position
//     PlcTask Inputs/Main.M19.nRawEncoderULINT <-> FB Inputs Channel 1/Position
//   tmo_motion Instance <-> Device 1 (EtherCAT)/Power (EK1200)/PLC Junction 2 (EK1122)/PLC Coupler 2 (EK1100)/PLC Junction 10 (EK1122)/PF1K4-WFS (EK1100)/PF1K4-EL7041-E1
//     PlcTask Inputs/Main.M18.bLimitBackwardEnable <-> STM Status/Status/Digital input 2
//     PlcTask Inputs/Main.M18.bLimitForwardEnable <-> STM Status/Status/Digital input 1
//   tmo_motion Instance <-> Device 1 (EtherCAT)/Power (EK1200)/PLC Junction 2 (EK1122)/PLC Coupler 2 (EK1100)/PLC Junction 7 (EK1122)/TM1K4-ATM (EK1100)/TM1K4-EL2004-E4
//     PlcTask Outputs/Main.M21.bBrakeRelease <-> Channel 1/Output
//   tmo_motion Instance <-> Device 1 (EtherCAT)/Power (EK1200)/PLC Junction 2 (EK1122)/PLC Coupler 2 (EK1100)/PLC Junction 7 (EK1122)/TM1K4-ATM (EK1100)/TM1K4-EL3314-E5
//     PlcTask Inputs/PRG_TM1K4.fbTM1K4.fbTempSensor1.bError <-> TC Inputs Channel 1/Status/Error
//     PlcTask Inputs/PRG_TM1K4.fbTM1K4.fbTempSensor1.bOverrange <-> TC Inputs Channel 1/Status/Overrange
//     PlcTask Inputs/PRG_TM1K4.fbTM1K4.fbTempSensor1.bUnderrange <-> TC Inputs Channel 1/Status/Underrange
//     PlcTask Inputs/PRG_TM1K4.fbTM1K4.fbTempSensor1.iRaw <-> TC Inputs Channel 1/Value
//   tmo_motion Instance <-> Device 1 (EtherCAT)/Power (EK1200)/PLC Junction 2 (EK1122)/PLC Coupler 2 (EK1100)/PLC Junction 7 (EK1122)/TM1K4-ATM (EK1100)/TM1K4-EL5042-E3
//     PlcTask Inputs/Main.M21.nRawEncoderULINT <-> FB Inputs Channel 1/Position
//     PlcTask Inputs/Main.M22.nRawEncoderULINT <-> FB Inputs Channel 2/Position
//   tmo_motion Instance <-> Device 1 (EtherCAT)/Power (EK1200)/PLC Junction 2 (EK1122)/PLC Coupler 2 (EK1100)/PLC Junction 7 (EK1122)/TM1K4-ATM (EK1100)/TM1K4-EL7041-E1
//     PlcTask Inputs/Main.M21.bLimitBackwardEnable <-> STM Status/Status/Digital input 2
//     PlcTask Inputs/Main.M21.bLimitForwardEnable <-> STM Status/Status/Digital input 1
//   tmo_motion Instance <-> Device 1 (EtherCAT)/Power (EK1200)/PLC Junction 2 (EK1122)/PLC Coupler 2 (EK1100)/PLC Junction 8 (EK1122)/EP3174-FWM-E2
//     PlcTask Inputs/PRG_PC5K4.fbFlowMeter.iRaw <-> AI Standard Channel 1/Value
//     PlcTask Inputs/PRG_SP1K4.fbFlowMeter.iRaw <-> AI Standard Channel 2/Value
//     PlcTask Inputs/PRG_ST4K4_TMO_TERM.fbFlowMeter.iRaw <-> AI Standard Channel 1/Value
//   tmo_motion Instance <-> Device 1 (EtherCAT)/Power (EK1200)/PLC Junction 2 (EK1122)/PLC Coupler 2 (EK1100)/PLC Junction 8 (EK1122)/IM5K4-PPM (EK1100)/IM5K4-EL2004-E3
//     PlcTask Outputs/Main.M17.bBrakeRelease <-> Channel 1/Output
//     PlcTask Outputs/PRG_IM5K4_PPM.fbIM5K4.fbGige.bGigePower <-> Channel 2/Output
//   tmo_motion Instance <-> Device 1 (EtherCAT)/Power (EK1200)/PLC Junction 2 (EK1122)/PLC Coupler 2 (EK1100)/PLC Junction 8 (EK1122)/IM5K4-PPM (EK1100)/IM5K4-EL3052-E5
//     PlcTask Inputs/PRG_IM5K4_PPM.fbIM5K4.fbFlowMeter.iRaw <-> AI Standard Channel 1/Value
//     PlcTask Inputs/PRG_PF1K4_WFS_TARGET.fbPF1K4.fbFlowMeter.iRaw <-> AI Standard Channel 1/Value
//     PlcTask Inputs/PRG_TM1K4.fbTM1K4.fbFlowMeter.iRaw <-> AI Standard Channel 1/Value
//   tmo_motion Instance <-> Device 1 (EtherCAT)/Power (EK1200)/PLC Junction 2 (EK1122)/PLC Coupler 2 (EK1100)/PLC Junction 8 (EK1122)/IM5K4-PPM (EK1100)/IM5K4-EL3062-E6
//     PlcTask Inputs/PRG_IM5K4_PPM.fbIM5K4.fbPowerMeter.iVoltageINT <-> AI Standard Channel 1/Value
//   tmo_motion Instance <-> Device 1 (EtherCAT)/Power (EK1200)/PLC Junction 2 (EK1122)/PLC Coupler 2 (EK1100)/PLC Junction 8 (EK1122)/IM5K4-PPM (EK1100)/IM5K4-EL3314-E4
//     PlcTask Inputs/PRG_IM5K4_PPM.fbIM5K4.fbPowerMeter.fbTempSensor.bError <-> TC Inputs Channel 1/Status/Error
//     PlcTask Inputs/PRG_IM5K4_PPM.fbIM5K4.fbPowerMeter.fbTempSensor.bOverrange <-> TC Inputs Channel 1/Status/Overrange
//     PlcTask Inputs/PRG_IM5K4_PPM.fbIM5K4.fbPowerMeter.fbTempSensor.bUnderrange <-> TC Inputs Channel 1/Status/Underrange
//     PlcTask Inputs/PRG_IM5K4_PPM.fbIM5K4.fbPowerMeter.fbTempSensor.iRaw <-> TC Inputs Channel 1/Value
//     PlcTask Inputs/PRG_IM5K4_PPM.fbIM5K4.fbYagTempSensor.bError <-> TC Inputs Channel 2/Status/Error
//     PlcTask Inputs/PRG_IM5K4_PPM.fbIM5K4.fbYagTempSensor.bOverrange <-> TC Inputs Channel 2/Status/Overrange
//     PlcTask Inputs/PRG_IM5K4_PPM.fbIM5K4.fbYagTempSensor.bUnderrange <-> TC Inputs Channel 2/Status/Underrange
//     PlcTask Inputs/PRG_IM5K4_PPM.fbIM5K4.fbYagTempSensor.iRaw <-> TC Inputs Channel 2/Value
//   tmo_motion Instance <-> Device 1 (EtherCAT)/Power (EK1200)/PLC Junction 2 (EK1122)/PLC Coupler 2 (EK1100)/PLC Junction 8 (EK1122)/IM5K4-PPM (EK1100)/IM5K4-EL4004-E7
//     PlcTask Outputs/PRG_IM5K4_PPM.fbIM5K4.fbGige.iIlluminatorINT <-> AO Outputs Channel 1/Analog output
//   tmo_motion Instance <-> Device 1 (EtherCAT)/Power (EK1200)/PLC Junction 2 (EK1122)/PLC Coupler 2 (EK1100)/PLC Junction 8 (EK1122)/IM5K4-PPM (EK1100)/IM5K4-EL5042-E2
//     PlcTask Inputs/Main.M17.nRawEncoderULINT <-> FB Inputs Channel 1/Position
//   tmo_motion Instance <-> Device 1 (EtherCAT)/Power (EK1200)/PLC Junction 2 (EK1122)/PLC Coupler 2 (EK1100)/PLC Junction 8 (EK1122)/IM5K4-PPM (EK1100)/IM5K4-EL7041-E1
//     PlcTask Inputs/Main.M17.bLimitBackwardEnable <-> STM Status/Status/Digital input 2
//     PlcTask Inputs/Main.M17.bLimitForwardEnable <-> STM Status/Status/Digital input 1
//   tmo_motion Instance <-> Device 1 (EtherCAT)/Power (EK1200)/PLC Junction 2 (EK1122)/PLC Coupler 2 (EK1100)/PLC Junction 8 (EK1122)/ST4K4-TERM (EP2338-0001)
//     PlcTask Inputs/PRG_ST4K4_TMO_TERM.ST4K4.i_xInsertedLS <-> Channel 4/Input
//     PlcTask Inputs/PRG_ST4K4_TMO_TERM.ST4K4.i_xRetractedLS <-> Channel 3/Input
//     PlcTask Outputs/PRG_ST4K4_TMO_TERM.ST4K4.q_xRetract_DO <-> Channel 9/Output
//   tmo_motion Instance <-> Device 1 (EtherCAT)/Power (EK1200)/PLC Junction 2 (EK1122)/PLC Coupler 2 (EK1100)/PLC Junction 9 (EK1122)/LI2K4-PA1K4 (EK1100)/LI2K4-EL5042-E2
//     PlcTask Inputs/Main.M45.nRawEncoderULINT <-> FB Inputs Channel 1/Position
//     PlcTask Inputs/Main.M46.nRawEncoderULINT <-> FB Inputs Channel 2/Position
//   tmo_motion Instance <-> Device 1 (EtherCAT)/Power (EK1200)/PLC Junction 2 (EK1122)/PLC Coupler 2 (EK1100)/PLC Junction 9 (EK1122)/LI2K4-PA1K4 (EK1100)/LI2K4X-EL7047-E3
//     PlcTask Inputs/Main.M46.bLimitBackwardEnable <-> STM Status/Status/Digital input 2
//     PlcTask Inputs/Main.M46.bLimitForwardEnable <-> STM Status/Status/Digital input 1
//   tmo_motion Instance <-> Device 1 (EtherCAT)/Power (EK1200)/PLC Junction 2 (EK1122)/PLC Coupler 2 (EK1100)/PLC Junction 9 (EK1122)/LI2K4-PA1K4 (EK1100)/LI2K4Y-EL7047-E1
//     PlcTask Inputs/Main.M45.bLimitBackwardEnable <-> STM Status/Status/Digital input 2
//     PlcTask Inputs/Main.M45.bLimitForwardEnable <-> STM Status/Status/Digital input 1
//   tmo_motion Instance <-> Device 1 (EtherCAT)/Power (EK1200)/PLC Junction 2 (EK1122)/PLC Coupler 2 (EK1100)/PLC Junction 9 (EK1122)/LI2K4-PA1K4 (EK1100)/PA1K4-PF-EL5042-E5
//     PlcTask Inputs/Main.M47.nRawEncoderULINT <-> FB Inputs Channel 1/Position
//   tmo_motion Instance <-> Device 1 (EtherCAT)/Power (EK1200)/PLC Junction 2 (EK1122)/PLC Coupler 2 (EK1100)/PLC Junction 9 (EK1122)/LI2K4-PA1K4 (EK1100)/PA1K4-PF-EL7047-E4
//     PlcTask Inputs/Main.M47.bLimitBackwardEnable <-> STM Status/Status/Digital input 2
//     PlcTask Inputs/Main.M47.bLimitForwardEnable <-> STM Status/Status/Digital input 1
//   tmo_motion Instance <-> Device 1 (EtherCAT)/Power (EK1200)/PLC Junction 2 (EK1122)/PLC Coupler 2 (EK1100)/PLC Junction 9 (EK1122)/SP1K4 Bottom Rail (EK1100)/FoilX-EL7041
//     PlcTask Inputs/Main.M33.bLimitBackwardEnable <-> STM Status/Status/Digital input 1
//     PlcTask Inputs/Main.M33.bLimitForwardEnable <-> STM Status/Status/Digital input 2
//   tmo_motion Instance <-> Device 1 (EtherCAT)/Power (EK1200)/PLC Junction 2 (EK1122)/PLC Coupler 2 (EK1100)/PLC Junction 9 (EK1122)/SP1K4 Bottom Rail (EK1100)/LensX_EL1004
//     PlcTask Inputs/PRG_SP1K4.bHallInput1 <-> Channel 1/Input
//     PlcTask Inputs/PRG_SP1K4.bHallInput2 <-> Channel 2/Input
//   tmo_motion Instance <-> Device 1 (EtherCAT)/Power (EK1200)/PLC Junction 2 (EK1122)/PLC Coupler 2 (EK1100)/PLC Junction 9 (EK1122)/SP1K4 Bottom Rail (EK1100)/YagTheta-EL7041
//     PlcTask Inputs/Main.M40.bLimitBackwardEnable <-> STM Status/Status/Digital input 2
//     PlcTask Inputs/Main.M40.bLimitForwardEnable <-> STM Status/Status/Digital input 1
//   tmo_motion Instance <-> Device 1 (EtherCAT)/Power (EK1200)/PLC Junction 2 (EK1122)/PLC Coupler 2 (EK1100)/PLC Junction 9 (EK1122)/SP1K4 Bottom Rail (EK1100)/YagX-EL7041
//     PlcTask Inputs/Main.M37.bLimitBackwardEnable <-> STM Status/Status/Digital input 1
//     PlcTask Inputs/Main.M37.bLimitForwardEnable <-> STM Status/Status/Digital input 2
//   tmo_motion Instance <-> Device 1 (EtherCAT)/Power (EK1200)/PLC Junction 2 (EK1122)/PLC Coupler 2 (EK1100)/PLC Junction 9 (EK1122)/SP1K4 Bottom Rail (EK1100)/YagY-EL7041
//     PlcTask Inputs/Main.M38.bLimitBackwardEnable <-> STM Status/Status/Digital input 2
//     PlcTask Inputs/Main.M38.bLimitForwardEnable <-> STM Status/Status/Digital input 1
//   tmo_motion Instance <-> Device 1 (EtherCAT)/Power (EK1200)/PLC Junction 2 (EK1122)/PLC Coupler 2 (EK1100)/PLC Junction 9 (EK1122)/SP1K4 Bottom Rail (EK1100)/YagZ-EL7041
//     PlcTask Inputs/Main.M39.bLimitBackwardEnable <-> STM Status/Status/Digital input 1
//     PlcTask Inputs/Main.M39.bLimitForwardEnable <-> STM Status/Status/Digital input 2
//   tmo_motion Instance <-> Device 1 (EtherCAT)/Power (EK1200)/PLC Junction 2 (EK1122)/PLC Coupler 2 (EK1100)/PLC Junction 9 (EK1122)/SP1K4 Bottom Rail (EK1100)/ZonePlateX-EL7041
//     PlcTask Inputs/Main.M34.bLimitBackwardEnable <-> STM Status/Status/Digital input 1
//     PlcTask Inputs/Main.M34.bLimitForwardEnable <-> STM Status/Status/Digital input 2
//   tmo_motion Instance <-> Device 1 (EtherCAT)/Power (EK1200)/PLC Junction 2 (EK1122)/PLC Coupler 2 (EK1100)/PLC Junction 9 (EK1122)/SP1K4 Bottom Rail (EK1100)/ZonePlateY-EL7041
//     PlcTask Inputs/Main.M35.bLimitBackwardEnable <-> STM Status/Status/Digital input 1
//     PlcTask Inputs/Main.M35.bLimitForwardEnable <-> STM Status/Status/Digital input 2
//   tmo_motion Instance <-> Device 1 (EtherCAT)/Power (EK1200)/PLC Junction 2 (EK1122)/PLC Coupler 2 (EK1100)/PLC Junction 9 (EK1122)/SP1K4 Bottom Rail (EK1100)/ZonePlateZ-EL7041
//     PlcTask Inputs/Main.M36.bLimitBackwardEnable <-> STM Status/Status/Digital input 2
//     PlcTask Inputs/Main.M36.bLimitForwardEnable <-> STM Status/Status/Digital input 1
//   tmo_motion Instance <-> Device 1 (EtherCAT)/Power (EK1200)/PLC Junction 2 (EK1122)/PLC Coupler 2 (EK1100)/PLC Junction 9 (EK1122)/SP1K4 Top Rail (EK1100)/FoilY-EL7041
//     PlcTask Inputs/Main.M44.bLimitBackwardEnable <-> STM Status/Status/Digital input 2
//     PlcTask Inputs/Main.M44.bLimitForwardEnable <-> STM Status/Status/Digital input 1
//   tmo_motion Instance <-> Device 1 (EtherCAT)/Power (EK1200)/PLC Junction 2 (EK1122)/PLC Coupler 2 (EK1100)/PLC Junction 9 (EK1122)/SP1K4 Top Rail (EK1100)/SP1K4-EL3202-E9A
//     PlcTask Inputs/PRG_SP1K4.SP1K4_ATT_RTD_01.bError <-> RTD Inputs Channel 1/Status/Error
//     PlcTask Inputs/PRG_SP1K4.SP1K4_ATT_RTD_02.bError <-> RTD Inputs Channel 2/Status/Error
//     PlcTask Inputs/PRG_SP1K4.SP1K4_ATT_RTD_01.bOverrange <-> RTD Inputs Channel 1/Status/Overrange
//     PlcTask Inputs/PRG_SP1K4.SP1K4_ATT_RTD_02.bOverrange <-> RTD Inputs Channel 2/Status/Overrange
//     PlcTask Inputs/PRG_SP1K4.SP1K4_ATT_RTD_01.bUnderrange <-> RTD Inputs Channel 1/Status/Underrange
//     PlcTask Inputs/PRG_SP1K4.SP1K4_ATT_RTD_02.bUnderrange <-> RTD Inputs Channel 2/Status/Underrange
//     PlcTask Inputs/PRG_SP1K4.SP1K4_ATT_RTD_01.iRaw <-> RTD Inputs Channel 1/Value
//     PlcTask Inputs/PRG_SP1K4.SP1K4_ATT_RTD_02.iRaw <-> RTD Inputs Channel 2/Value
//   tmo_motion Instance <-> Device 1 (EtherCAT)/Power (EK1200)/PLC Junction 2 (EK1122)/PLC Coupler 2 (EK1100)/PLC Junction 9 (EK1122)/SP1K4 Top Rail (EK1100)/SP1K4-EL5042-E8
//     PlcTask Inputs/Main.M38.nRawEncoderULINT <-> FB Inputs Channel 1/Position
//   tmo_motion Instance <-> Device 1 (EtherCAT)/Power (EK1200)/PLC Junction 2 (EK1122)/PLC Coupler 2 (EK1100)/PLC Junction 9 (EK1122)/SP1K4 Top Rail (EK1100)/SP1K4-TL1-EL1124
//     PlcTask Inputs/PRG_SP1K4.bTL1High <-> Channel 1/Input
//     PlcTask Inputs/PRG_SP1K4.bTL1Low <-> Channel 2/Input
//   tmo_motion Instance <-> Device 1 (EtherCAT)/Power (EK1200)/PLC Junction 2 (EK1122)/PLC Coupler 2 (EK1100)/PLC Junction 9 (EK1122)/SP1K4 Top Rail (EK1100)/SP1K4-TL2-EL1124
//     PlcTask Inputs/PRG_SP1K4.bTL2High <-> Channel 1/Input
//     PlcTask Inputs/PRG_SP1K4.bTL2Low <-> Channel 2/Input
//   tmo_motion Instance <-> Device 1 (EtherCAT)/Power (EK1200)/PMPS_FFO
//     PlcTask Outputs/GVL_PMPS.fbFastFaultOutput1.q_xFastFaultOut <-> Channel 1/Output
//     PlcTask Outputs/GVL_PMPS.fbFastFaultOutput2.q_xFastFaultOut <-> Channel 2/Output
//   tmo_motion Instance <-> Device 1 (EtherCAT)/Power (EK1200)/PMPS_PRE
//     PlcTask Inputs/PRG_3_PMPS_POST.fbArbiterIO.i_stCurrentBP <-> IO Inputs/CurrentBP
//     PlcTask Inputs/PRG_3_PMPS_POST.fbArbiterIO.xTxPDO_state <-> SYNC Inputs/TxPDO state
//     PlcTask Inputs/PRG_3_PMPS_POST.fbArbiterIO.xTxPDO_toggle <-> SYNC Inputs/TxPDO toggle
//     PlcTask Outputs/GVL_PMPS.PMPS_ST4K4_IN <-> IO Outputs/bST4K4_IN
//     PlcTask Outputs/GVL_PMPS.PMPS_ST4K4_OUT <-> IO Outputs/bST4K4_OUT
//     PlcTask Outputs/PRG_3_PMPS_POST.fbArbiterIO.q_stRequestedBP <-> IO Outputs/RequestedBP
//   tmo_motion Instance <-> NC-Task 1 SAF/Axes/Axis 1 AL1K4-L2SI-MMS
//     PlcTask Inputs/Main.M1.Axis.NcToPlc <-> Outputs/ToPlc
//     PlcTask Outputs/Main.M1.Axis.PlcToNc <-> Inputs/FromPlc
//   tmo_motion Instance <-> NC-Task 1 SAF/Axes/Axis 15 IM3K4-PPM-MMS
//     PlcTask Inputs/Main.M15.Axis.NcToPlc <-> Outputs/ToPlc
//     PlcTask Outputs/Main.M15.Axis.PlcToNc <-> Inputs/FromPlc
//   tmo_motion Instance <-> NC-Task 1 SAF/Axes/Axis 16 IM4K4-PPM-MMS
//     PlcTask Inputs/Main.M16.Axis.NcToPlc <-> Outputs/ToPlc
//     PlcTask Outputs/Main.M16.Axis.PlcToNc <-> Inputs/FromPlc
//   tmo_motion Instance <-> NC-Task 1 SAF/Axes/Axis 17 IM5K4-PPM-MMS
//     PlcTask Inputs/Main.M17.Axis.NcToPlc <-> Outputs/ToPlc
//     PlcTask Outputs/Main.M17.Axis.PlcToNc <-> Inputs/FromPlc
//   tmo_motion Instance <-> NC-Task 1 SAF/Axes/Axis 18 PF1K4-WFS_TARGET-MMS-Y
//     PlcTask Inputs/Main.M18.Axis.NcToPlc <-> Outputs/ToPlc
//     PlcTask Outputs/Main.M18.Axis.PlcToNc <-> Inputs/FromPlc
//   tmo_motion Instance <-> NC-Task 1 SAF/Axes/Axis 19 PF1K4-WFS_TARGET-MMS-Z
//     PlcTask Inputs/Main.M19.Axis.NcToPlc <-> Outputs/ToPlc
//     PlcTask Outputs/Main.M19.Axis.PlcToNc <-> Inputs/FromPlc
//   tmo_motion Instance <-> NC-Task 1 SAF/Axes/Axis 2
//     PlcTask Inputs/Main.M2.Axis.NcToPlc <-> Outputs/ToPlc
//     PlcTask Outputs/Main.M2.Axis.PlcToNc <-> Inputs/FromPlc
//   tmo_motion Instance <-> NC-Task 1 SAF/Axes/Axis 20 LI1K4-IP1-MMS
//     PlcTask Inputs/Main.M20.Axis.NcToPlc <-> Outputs/ToPlc
//     PlcTask Outputs/Main.M20.Axis.PlcToNc <-> Inputs/FromPlc
//   tmo_motion Instance <-> NC-Task 1 SAF/Axes/Axis 21 TM1K4-MMS-Y
//     PlcTask Inputs/Main.M21.Axis.NcToPlc <-> Outputs/ToPlc
//     PlcTask Outputs/Main.M21.Axis.PlcToNc <-> Inputs/FromPlc
//   tmo_motion Instance <-> NC-Task 1 SAF/Axes/Axis 22 TM1K4-MMS-X
//     PlcTask Inputs/Main.M22.Axis.NcToPlc <-> Outputs/ToPlc
//     PlcTask Outputs/Main.M22.Axis.PlcToNc <-> Inputs/FromPlc
//   tmo_motion Instance <-> NC-Task 1 SAF/Axes/Axis 27 IM6K4-PPM-MMS
//     PlcTask Inputs/Main.M27.Axis.NcToPlc <-> Outputs/ToPlc
//     PlcTask Outputs/Main.M27.Axis.PlcToNc <-> Inputs/FromPlc
//   tmo_motion Instance <-> NC-Task 1 SAF/Axes/Axis 28 PF2K4-WFS_TARGET-MMS-Y
//     PlcTask Inputs/Main.M28.Axis.NcToPlc <-> Outputs/ToPlc
//     PlcTask Outputs/Main.M28.Axis.PlcToNc <-> Inputs/FromPlc
//   tmo_motion Instance <-> NC-Task 1 SAF/Axes/Axis 29 PF2K4-WFS_TARGET-MMS-Z
//     PlcTask Inputs/Main.M29.Axis.NcToPlc <-> Outputs/ToPlc
//     PlcTask Outputs/Main.M29.Axis.PlcToNc <-> Inputs/FromPlc
//   tmo_motion Instance <-> NC-Task 1 SAF/Axes/Axis 3
//     PlcTask Inputs/Main.M3.Axis.NcToPlc <-> Outputs/ToPlc
//     PlcTask Outputs/Main.M3.Axis.PlcToNc <-> Inputs/FromPlc
//   tmo_motion Instance <-> NC-Task 1 SAF/Axes/Axis 30 TM2K4-MMS-Y
//     PlcTask Inputs/Main.M30.Axis.NcToPlc <-> Outputs/ToPlc
//     PlcTask Outputs/Main.M30.Axis.PlcToNc <-> Inputs/FromPlc
//   tmo_motion Instance <-> NC-Task 1 SAF/Axes/Axis 31 TM2K4-MMS-X
//     PlcTask Inputs/Main.M31.Axis.NcToPlc <-> Outputs/ToPlc
//     PlcTask Outputs/Main.M31.Axis.PlcToNc <-> Inputs/FromPlc
//   tmo_motion Instance <-> NC-Task 1 SAF/Axes/Axis 4
//     PlcTask Inputs/Main.M4.Axis.NcToPlc <-> Outputs/ToPlc
//     PlcTask Outputs/Main.M4.Axis.PlcToNc <-> Inputs/FromPlc
//   tmo_motion Instance <-> NC-Task 1 SAF/Axes/Axis 45 LI2K4-MMS-Y
//     PlcTask Inputs/Main.M45.Axis.NcToPlc <-> Outputs/ToPlc
//     PlcTask Outputs/Main.M45.Axis.PlcToNc <-> Inputs/FromPlc
//   tmo_motion Instance <-> NC-Task 1 SAF/Axes/Axis 46 LI2K4-MMS-X
//     PlcTask Inputs/Main.M46.Axis.NcToPlc <-> Outputs/ToPlc
//     PlcTask Outputs/Main.M46.Axis.PlcToNc <-> Inputs/FromPlc
//   tmo_motion Instance <-> NC-Task 1 SAF/Axes/Axis 5
//     PlcTask Inputs/Main.M5.Axis.NcToPlc <-> Outputs/ToPlc
//     PlcTask Outputs/Main.M5.Axis.PlcToNc <-> Inputs/FromPlc
//   tmo_motion Instance <-> NC-Task 1 SAF/Axes/Axis 6 IM1K4-XTES-MMS
//     PlcTask Inputs/Main.M6.Axis.NcToPlc <-> Outputs/ToPlc
//     PlcTask Outputs/Main.M6.Axis.PlcToNc <-> Inputs/FromPlc
//   tmo_motion Instance <-> NC-Task 1 SAF/Axes/Axis 7 IM1K4-XTES-CLZ
//     PlcTask Inputs/Main.M7.Axis.NcToPlc <-> Outputs/ToPlc
//     PlcTask Outputs/Main.M7.Axis.PlcToNc <-> Inputs/FromPlc
//   tmo_motion Instance <-> NC-Task 1 SAF/Axes/Axis 8 IM1K4-XTES-CLF
//     PlcTask Inputs/Main.M8.Axis.NcToPlc <-> Outputs/ToPlc
//     PlcTask Outputs/Main.M8.Axis.PlcToNc <-> Inputs/FromPlc
//   tmo_motion Instance <-> NC-Task 1 SAF/Axes/Axis 9 IM2K4-PPM-MMS
//     PlcTask Inputs/Main.M9.Axis.NcToPlc <-> Outputs/ToPlc
//     PlcTask Outputs/Main.M9.Axis.PlcToNc <-> Inputs/FromPlc
//   tmo_motion Instance <-> NC-Task 1 SAF/Axes/FoilX
//     PlcTask Inputs/Main.M33.Axis.NcToPlc <-> Outputs/ToPlc
//     PlcTask Outputs/Main.M33.Axis.PlcToNc <-> Inputs/FromPlc
//   tmo_motion Instance <-> NC-Task 1 SAF/Axes/FoilY
//     PlcTask Inputs/Main.M44.Axis.NcToPlc <-> Outputs/ToPlc
//     PlcTask Outputs/Main.M44.Axis.PlcToNc <-> Inputs/FromPlc
//   tmo_motion Instance <-> NC-Task 1 SAF/Axes/LensX
//     PlcTask Inputs/Main.M32.Axis.NcToPlc <-> Outputs/ToPlc
//     PlcTask Outputs/Main.M32.Axis.PlcToNc <-> Inputs/FromPlc
//   tmo_motion Instance <-> NC-Task 1 SAF/Axes/PA1K4-PF-MMS
//     PlcTask Inputs/Main.M47.Axis.NcToPlc <-> Outputs/ToPlc
//     PlcTask Outputs/Main.M47.Axis.PlcToNc <-> Inputs/FromPlc
//   tmo_motion Instance <-> NC-Task 1 SAF/Axes/SL1K4-BOTTOM-M10
//     PlcTask Inputs/Main.M10.Axis.NcToPlc <-> Outputs/ToPlc
//     PlcTask Outputs/Main.M10.Axis.PlcToNc <-> Inputs/FromPlc
//   tmo_motion Instance <-> NC-Task 1 SAF/Axes/SL1K4-NORTH-M12
//     PlcTask Inputs/Main.M12.Axis.NcToPlc <-> Outputs/ToPlc
//     PlcTask Outputs/Main.M12.Axis.PlcToNc <-> Inputs/FromPlc
//   tmo_motion Instance <-> NC-Task 1 SAF/Axes/SL1K4-SOUTH-M13
//     PlcTask Inputs/Main.M13.Axis.NcToPlc <-> Outputs/ToPlc
//     PlcTask Outputs/Main.M13.Axis.PlcToNc <-> Inputs/FromPlc
//   tmo_motion Instance <-> NC-Task 1 SAF/Axes/SL1K4-TOP-M11
//     PlcTask Inputs/Main.M11.Axis.NcToPlc <-> Outputs/ToPlc
//     PlcTask Outputs/Main.M11.Axis.PlcToNc <-> Inputs/FromPlc
//   tmo_motion Instance <-> NC-Task 1 SAF/Axes/ST1K4-TEST
//     PlcTask Inputs/Main.M14.Axis.NcToPlc <-> Outputs/ToPlc
//     PlcTask Outputs/Main.M14.Axis.PlcToNc <-> Inputs/FromPlc
//   tmo_motion Instance <-> NC-Task 1 SAF/Axes/Thorlab-LenX
//     PlcTask Inputs/Main.M43.Axis.NcToPlc <-> Outputs/ToPlc
//     PlcTask Outputs/Main.M43.Axis.PlcToNc <-> Inputs/FromPlc
//   tmo_motion Instance <-> NC-Task 1 SAF/Axes/Thorlabs1
//     PlcTask Inputs/Main.M41.Axis.NcToPlc <-> Outputs/ToPlc
//     PlcTask Outputs/Main.M41.Axis.PlcToNc <-> Inputs/FromPlc
//   tmo_motion Instance <-> NC-Task 1 SAF/Axes/Thorlabs2
//     PlcTask Inputs/Main.M42.Axis.NcToPlc <-> Outputs/ToPlc
//     PlcTask Outputs/Main.M42.Axis.PlcToNc <-> Inputs/FromPlc
//   tmo_motion Instance <-> NC-Task 1 SAF/Axes/YagTheta
//     PlcTask Inputs/Main.M40.Axis.NcToPlc <-> Outputs/ToPlc
//     PlcTask Outputs/Main.M40.Axis.PlcToNc <-> Inputs/FromPlc
//   tmo_motion Instance <-> NC-Task 1 SAF/Axes/YagX
//     PlcTask Inputs/Main.M37.Axis.NcToPlc <-> Outputs/ToPlc
//     PlcTask Outputs/Main.M37.Axis.PlcToNc <-> Inputs/FromPlc
//   tmo_motion Instance <-> NC-Task 1 SAF/Axes/YagY
//     PlcTask Inputs/Main.M38.Axis.NcToPlc <-> Outputs/ToPlc
//     PlcTask Outputs/Main.M38.Axis.PlcToNc <-> Inputs/FromPlc
//   tmo_motion Instance <-> NC-Task 1 SAF/Axes/YagZ
//     PlcTask Inputs/Main.M39.Axis.NcToPlc <-> Outputs/ToPlc
//     PlcTask Outputs/Main.M39.Axis.PlcToNc <-> Inputs/FromPlc
//   tmo_motion Instance <-> NC-Task 1 SAF/Axes/ZonePlateX
//     PlcTask Inputs/Main.M34.Axis.NcToPlc <-> Outputs/ToPlc
//     PlcTask Outputs/Main.M34.Axis.PlcToNc <-> Inputs/FromPlc
//   tmo_motion Instance <-> NC-Task 1 SAF/Axes/ZonePlateY
//     PlcTask Inputs/Main.M35.Axis.NcToPlc <-> Outputs/ToPlc
//     PlcTask Outputs/Main.M35.Axis.PlcToNc <-> Inputs/FromPlc
//   tmo_motion Instance <-> NC-Task 1 SAF/Axes/ZonePlateZ
//     PlcTask Inputs/Main.M36.Axis.NcToPlc <-> Outputs/ToPlc
//     PlcTask Outputs/Main.M36.Axis.PlcToNc <-> Inputs/FromPlc

// ---- DUTs/ENUM_SolidAttenuator_States.TcDUT
{attribute 'qualified_only'}
{attribute 'strict'}
TYPE ENUM_SolidAttenuator_States :
(
    Unknown := 0,
    OUT := 1,
    Target1 := 2,
    Target2 := 3,
    Target3 := 4,
    Target4 := 5,
    Target5 := 6,
    Target6 := 7, // add four more targets on 9-9-25
    Target7 := 8,
    Target8 := 9,
    Target9 := 10

)UINT;
END_TYPE

// ---- DUTs/ENUM_LaserCoupling_States.TcDUT
{attribute 'qualified_only'}
{attribute 'strict'}
TYPE ENUM_LaserCoupling_States :
(
    Unknown := 0,
    OUT := 1,
    Mirror1 := 2

)UINT;
END_TYPE

// ---- DUTs/ENUM_Sample_Calibration_States.TcDUT
{attribute 'qualified_only'}
{attribute 'strict'}
TYPE ENUM_Sample_Calibration_States :
(
    Unknown := 0,
    OUT := 1,
    Target1 := 2,
    Target2 := 3,
    Target3 := 4,
    Target4 := 5,
    Target5 := 6
//    Target6 := 7,
//    Target7 := 8

)UINT;
END_TYPE

// ---- DUTs/ENUM_ZonePlate_States.TcDUT
{attribute 'qualified_only'}
TYPE ENUM_ZonePlate_States :
(
  // Third version of targets paddle 3
    Unknown := 0,
    OUT := 1,
    Target1b := 2,
    Target5a := 3,
    Target4b := 4,
    Target5b := 5,
    Target3b := 6,
    Target2b := 7,
    Target1a := 8,
    Target2a := 9,
    Target6b := 10,
    Target7b := 11,
    Target6a := 12,
    Target7a := 13,
    Target3a := 14,
    Target4a := 15
) UINT;
END_TYPE
    // first version of targets paddle 1
{*   FZP860_1 := 3,   //Ne1
    FZP860_2 := 4,   //Ne2
    FZP860_3 := 5,   //Ne3
    FZP750_1 := 6,   //3w1
    FZP750_2 := 7,   //3w2
    FZP530_1 := 8,   //o1
    FZP530_2 := 9,   //o2
    FZP460_1 := 10,   //Ti1
    FZP460_2 := 11,   //Ti2
    FZP410_1 := 12,   //N1
    FZP410_2 := 13,   //N2
    FZP290_1 := 14,   // C1
    FZP290_2 := 15   //C2
//	FZP250_1 := 16    //w1

    //second version of targets paddle 2
    FZP530_1 := 3,
    FZP806 := 4,
    FZP530_2 := 5,
    FZP1212_1 := 6,
    FZP404_1212_1 := 7,
    FZP262_524 := 8,
    FZP404_1212_2 := 9,
    FZP400_1 := 10,
    FZP290 := 11,
    FZP400_2 := 12,
    FZP350 := 13,
    FZP1212_2 := 14,
    FZP875 := 15
*}

// ---- DUTs/E_HomeState.TcDUT
TYPE E_HomeState :
(
	H_READY,
	H_INIT,
	H_RESET_LL,
	H_RESET_HL,
	H_ENABLE,
	H_MOVING,
	H_KEEP_MOVING,
	H_CHECK,
	H_RESET,
	H_SET_POS,
	H_ERROR,
	H_WRITE_LL,
	H_WRITE_HL,
	H_DONE
	
) UDINT;
END_TYPE

// ---- POUs/TM1K4/ENUM_TM1K4_States.TcDUT
{attribute 'qualified_only'}
TYPE ENUM_TM1K4_States :
(
    // Adapted from ENUM_ATM_States to add TARGET6

    Unknown := 0,
    OUT := 1,
    TARGET1a := 2,
    TARGET1b := 3,
    TARGET2a := 4,
    TARGET2b := 5,
    TARGET3a := 6,
    TARGET3b := 7,
    YAG := 8,
    DIODE := 9
) UINT;
END_TYPE

// ---- POUs/TM2K4/ENUM_TM2K4_States.TcDUT
{attribute 'qualified_only'}
TYPE ENUM_TM2K4_States :
(
    // Adapted from ENUM_ATM_States to add TARGET6

    Unknown := 0,
    OUT := 1,
    TARGET1a := 2,
    TARGET1b := 3,
    TARGET2a := 4,
    TARGET2b := 5,
    TARGET3a := 6,
    TARGET3b := 7,
    YAG := 8,
    DIODE := 9

) UINT;
END_TYPE

// ---- GVLs/GVL_PMPS.TcGVL
VAR_GLOBAL

    // Arbiter linked to the FFO and the MPS
    {attribute 'pytmc' := 'pv: PLC:TMO:MOTION:ARB:01'}
    fbArbiter: FB_Arbiter(1);

     // Arbiter linked to the FFO and the MPS
    {attribute 'pytmc' := 'pv: PLC:TMO:MOTION:ARB:02'}
    fbArbiter2: FB_Arbiter(2);

    // Fast fault for before ST4K4 (Most Devices)
    {attribute 'pytmc' := 'pv: PLC:TMO:MOTION:FFO:01'}
    {attribute 'TcLinkTo' := '.q_xFastFaultOut:=TIIB[PMPS_FFO]^Channel 1^Output'}
    fbFastFaultOutput1: FB_HardwareFFOutput := (bAutoReset := TRUE, i_sNetID:='172.21.92.73.1.1');
    // Fast fault for after ST4K4 (Basically just DREAM)
    {attribute 'pytmc' := 'pv: PLC:TMO:MOTION:FFO:02'}
    {attribute 'TcLinkTo' := '.q_xFastFaultOut:=TIIB[PMPS_FFO]^Channel 2^Output'}
    fbFastFaultOutput2: FB_HardwareFFOutput := (bAutoReset := TRUE, i_sNetID:='172.21.92.73.1.1');

    {attribute 'TcLinkTo' := 'TIIB[PMPS_PRE]^IO Outputs^bST4K4_IN'}
    PMPS_ST4K4_IN AT%Q* : BOOL;
    {attribute 'TcLinkTo' := 'TIIB[PMPS_PRE]^IO Outputs^bST4K4_OUT'}
    PMPS_ST4K4_OUT AT%Q* : BOOL;
END_VAR

// ---- GVLs/GVL_TcGVL.TcGVL
{attribute 'qualified_only'}
VAR_GLOBAL
    ePF1K4State: E_WFS_States;
    ePF2K4State:E_WFS_States;
    eSP1K4ATT:ENUM_SolidAttenuator_States;
    eSP1K4FZP:ENUM_ZonePlate_States;

END_VAR

// ---- GVLs/Main.TcGVL
{attribute 'qualified_only'}
VAR_GLOBAL
    // AL1K4-L2SI: 1 Axis
    {attribute 'pytmc' := 'pv: AL1K4:L2SI:MMS'}
    {attribute 'TcLinkTo' := '.bLimitForwardEnable  := TIIB[AL1K4-EL7041-E1]^STM Status^Status^Digital input 1;
                              .bLimitBackwardEnable := TIIB[AL1K4-EL7041-E1]^STM Status^Status^Digital input 2;
                              .bBrakeRelease        := TIIB[AL1K4-EL2004-E3]^Channel 1^Output;
                              .nRawEncoderULINT     := TIIB[AL1K4-EL5042-E2]^FB Inputs Channel 1^Position'}
    M1: ST_MotionStage := (sName := 'AL1K4:L2SI:MMS');

    // SPARE: 7 Axes (formerly AT1K4-SOLID and IM1K4-XTES)
    M2: ST_MotionStage;
    M3: ST_MotionStage;
    M4: ST_MotionStage;
    M5: ST_MotionStage;
    M6: ST_MotionStage;
    M7: ST_MotionStage;
    M8: ST_MotionStage;

    // IM2K4-PPM: 1 Axis
    {attribute 'pytmc' := 'pv: IM2K4:PPM:MMS'}
    {attribute 'TcLinkTo' := '.bLimitForwardEnable  := TIIB[IM2K4-EL7041-E1]^STM Status^Status^Digital input 1;
                              .bLimitBackwardEnable := TIIB[IM2K4-EL7041-E1]^STM Status^Status^Digital input 2;
                              .bBrakeRelease        := TIIB[IM2K4-EL2004-E3]^Channel 1^Output;
                              .nRawEncoderULINT     := TIIB[IM2K4-EL5042-E2]^FB Inputs Channel 1^Position'}
    M9: ST_MotionStage := (sName := 'IM2K4:PPM:MMS');

    // SL1K4-SCATTER: 4 Axes
    {attribute 'pytmc' := 'pv: SL1K4:SCATTER:MMS:BOTTOM'}
    {attribute 'TcLinkTo' := '.bLimitForwardEnable  := TIIB[SL1K4-EL7031-E1]^STM Status^Status^Digital input 2;
                              .bLimitBackwardEnable := TIIB[SL1K4-EL7031-E1]^STM Status^Status^Digital input 1;
                              .nRawEncoderUINT      := TIIB[SL1K4-EL5101-E2]^ENC Status compact^Counter value'}
    M10: ST_MotionStage := (sName := 'SL1K4:SCATTER:MMS:BOTTOM');
    {attribute 'pytmc' := 'pv: SL1K4:SCATTER:MMS:TOP'}
    {attribute 'TcLinkTo' := '.bLimitForwardEnable  := TIIB[SL1K4-EL7031-E3]^STM Status^Status^Digital input 2;
                              .bLimitBackwardEnable := TIIB[SL1K4-EL7031-E3]^STM Status^Status^Digital input 1;
                              .nRawEncoderUINT      := TIIB[SL1K4-EL5101-E4]^ENC Status compact^Counter value'}
    M11: ST_MotionStage := (sName := 'SL1K4:SCATTER:MMS:TOP');
    {attribute 'pytmc' := 'pv: SL1K4:SCATTER:MMS:NORTH'}
    {attribute 'TcLinkTo' := '.bLimitForwardEnable  := TIIB[SL1K4-EL7031-E5]^STM Status^Status^Digital input 1;
                              .bLimitBackwardEnable := TIIB[SL1K4-EL7031-E5]^STM Status^Status^Digital input 2;
                              .nRawEncoderUINT      := TIIB[SL1K4-EL5101-E6]^ENC Status compact^Counter value'}
    M12: ST_MotionStage := (sName := 'SL1K4:SCATTER:MMS:NORTH');
    {attribute 'pytmc' := 'pv: SL1K4:SCATTER:MMS:SOUTH'}
    {attribute 'TcLinkTo' := '.bLimitForwardEnable  := TIIB[SL1K4-EL7031-E7]^STM Status^Status^Digital input 1;
                              .bLimitBackwardEnable := TIIB[SL1K4-EL7031-E7]^STM Status^Status^Digital input 2;
                              .nRawEncoderUINT      := TIIB[SL1K4-EL5101-E8]^ENC Status compact^Counter value'}
    M13: ST_MotionStage := (sName := 'SL1K4:SCATTER:MMS:SOUTH');

    // SPARE: 1 Axis (formerly ST1K4-TEST)
    M14: ST_MotionStage;

    // IM3K4-PPM: 1 Axis
    {attribute 'pytmc' := 'pv: IM3K4:PPM:MMS'}
    {attribute 'TcLinkTo' := '.bLimitForwardEnable  := TIIB[IM3K4-EL7041-E1]^STM Status^Status^Digital input 1;
                              .bLimitBackwardEnable := TIIB[IM3K4-EL7041-E1]^STM Status^Status^Digital input 2;
                              .bBrakeRelease        := TIIB[IM3K4-EL2004-E3]^Channel 1^Output;
                              .nRawEncoderULINT     := TIIB[IM3K4-EL5042-E2]^FB Inputs Channel 1^Position'}
    M15: ST_MotionStage := (sName := 'IM3K4:PPM:MMS');
    // IM4K4-PPM: 1 Axis
    {attribute 'pytmc' := 'pv: IM4K4:PPM:MMS'}
    {attribute 'TcLinkTo' := '.bLimitForwardEnable  := TIIB[IM4K4-EL7041-E1]^STM Status^Status^Digital input 1;
                              .bLimitBackwardEnable := TIIB[IM4K4-EL7041-E1]^STM Status^Status^Digital input 2;
                              .bBrakeRelease        := TIIB[IM4K4-EL2004-E3]^Channel 1^Output;
                              .nRawEncoderULINT     := TIIB[IM4K4-EL5042-E2]^FB Inputs Channel 1^Position'}
    M16: ST_MotionStage := (sName := 'IM4K4:PPM:MMS');

